# B&R Automation Studio project TD52 (part 16)

```c
/* Source: dspcon.f */
#define dspcon FORTRAN_WRAPPER(dspcon)
extern void dspcon(
    char   *uplo,
    ptrdiff_t *n,
    double *ap,
    ptrdiff_t *ipiv,
    double *anorm,
    double *rcond,
    double *work,
    ptrdiff_t *iwork,
    ptrdiff_t *info
);

/* Source: dspev.f */
#define dspev FORTRAN_WRAPPER(dspev)
extern void dspev(
    char   *jobz,
    char   *uplo,
    ptrdiff_t *n,
    double *ap,
    double *w,
    double *z,
    ptrdiff_t *ldz,
    double *work,
    ptrdiff_t *info
);

/* Source: dspevd.f */
#define dspevd FORTRAN_WRAPPER(dspevd)
extern void dspevd(
    char   *jobz,
    char   *uplo,
    ptrdiff_t *n,
    double *ap,
    double *w,
    double *z,
    ptrdiff_t *ldz,
    double *work,
    ptrdiff_t *lwork,
    ptrdiff_t *iwork,
    ptrdiff_t *liwork,
    ptrdiff_t *info
);

/* Source: dspevx.f */
#define dspevx FORTRAN_WRAPPER(dspevx)
extern void dspevx(
    char   *jobz,
    char   *range,
    char   *uplo,
    ptrdiff_t *n,
    double *ap,
    double *vl,
    double *vu,
    ptrdiff_t *il,
    ptrdiff_t *iu,
    double *abstol,
    ptrdiff_t *m,
    double *w,
    double *z,
    ptrdiff_t *ldz,
    double *work,
    ptrdiff_t *iwork,
    ptrdiff_t *ifail,
    ptrdiff_t *info
);

/* Source: dspgst.f */
#define dspgst FORTRAN_WRAPPER(dspgst)
extern void dspgst(
    ptrdiff_t *itype,
    char   *uplo,
    ptrdiff_t *n,
    double *ap,
    double *bp,
    ptrdiff_t *info
);

/* Source: dspgv.f */
#define dspgv FORTRAN_WRAPPER(dspgv)
extern void dspgv(
    ptrdiff_t *itype,
    char   *jobz,
    char   *uplo,
    ptrdiff_t *n,
    double *ap,
    double *bp,
    double *w,
    double *z,
    ptrdiff_t *ldz,
    double *work,
    ptrdiff_t *info
);

/* Source: dspgvd.f */
#define dspgvd FORTRAN_WRAPPER(dspgvd)
extern void dspgvd(
    ptrdiff_t *itype,
    char   *jobz,
    char   *uplo,
    ptrdiff_t *n,
    double *ap,
    double *bp,
    double *w,
    double *z,
    ptrdiff_t *ldz,
    double *work,
    ptrdiff_t *lwork,
    ptrdiff_t *iwork,
    ptrdiff_t *liwork,
    ptrdiff_t *info
);

/* Source: dspgvx.f */
#define dspgvx FORTRAN_WRAPPER(dspgvx)
extern void dspgvx(
    ptrdiff_t *itype,
    char   *jobz,
    char   *range,
    char   *uplo,
    ptrdiff_t *n,
    double *ap,
    double *bp,
    double *vl,
    double *vu,
    ptrdiff_t *il,
    ptrdiff_t *iu,
    double *abstol,
    ptrdiff_t *m,
    double *w,
    double *z,
    ptrdiff_t *ldz,
    double *work,
    ptrdiff_t *iwork,
    ptrdiff_t *ifail,
    ptrdiff_t *info
);

/* Source: dsposv.f */
#define dsposv FORTRAN_WRAPPER(dsposv)
extern void dsposv(
    char   *uplo,
    ptrdiff_t *n,
    ptrdiff_t *nrhs,
    double *a,
    ptrdiff_t *lda,
    double *b,
    ptrdiff_t *ldb,
    double *x,
    ptrdiff_t *ldx,
    double *work,
    float  *swork,
    ptrdiff_t *iter,
    ptrdiff_t *info
);

/* Source: dsprfs.f */
#define dsprfs FORTRAN_WRAPPER(dsprfs)
extern void dsprfs(
    char   *uplo,
    ptrdiff_t *n,
    ptrdiff_t *nrhs,
    double *ap,
    double *afp,
    ptrdiff_t *ipiv,
    double *b,
    ptrdiff_t *ldb,
    double *x,
    ptrdiff_t *ldx,
    double *ferr,
    double *berr,
    double *work,
    ptrdiff_t *iwork,
    ptrdiff_t *info
);

/* Source: dspsv.f */
#define dspsv FORTRAN_WRAPPER(dspsv)
extern void dspsv(
    char   *uplo,
    ptrdiff_t *n,
    ptrdiff_t *nrhs,
    double *ap,
    ptrdiff_t *ipiv,
    double *b,
    ptrdiff_t *ldb,
    ptrdiff_t *info
);

/* Source: dspsvx.f */
#define dspsvx FORTRAN_WRAPPER(dspsvx)
extern void dspsvx(
    char   *fact,
    char   *uplo,
    ptrdiff_t *n,
    ptrdiff_t *nrhs,
    double *ap,
    double *afp,
    ptrdiff_t *ipiv,
    double *b,
    ptrdiff_t *ldb,
    double *x,
    ptrdiff_t *ldx,
    double *rcond,
    double *ferr,
    double *berr,
    double *work,
    ptrdiff_t *iwork,
    ptrdiff_t *info
);

/* Source: dsptrd.f */
#define dsptrd FORTRAN_WRAPPER(dsptrd)
extern void dsptrd(
    char   *uplo,
    ptrdiff_t *n,
    double *ap,
    double *d,
    double *e,
    double *tau,
    ptrdiff_t *info
);

/* Source: dsptrf.f */
#define dsptrf FORTRAN_WRAPPER(dsptrf)
extern void dsptrf(
    char   *uplo,
    ptrdiff_t *n,
    double *ap,
    ptrdiff_t *ipiv,
    ptrdiff_t *info
);

/* Source: dsptri.f */
#define dsptri FORTRAN_WRAPPER(dsptri)
extern void dsptri(
    char   *uplo,
    ptrdiff_t *n,
    double *ap,
    ptrdiff_t *ipiv,
    double *work,
    ptrdiff_t *info
);

/* Source: dsptrs.f */
#define dsptrs FORTRAN_WRAPPER(dsptrs)
extern void dsptrs(
    char   *uplo,
    ptrdiff_t *n,
    ptrdiff_t *nrhs,
    double *ap,
    ptrdiff_t *ipiv,
    double *b,
    ptrdiff_t *ldb,
    ptrdiff_t *info
);

/* Source: dstebz.f */
#define dstebz FORTRAN_WRAPPER(dstebz)
extern void dstebz(
    char   *range,
    char   *order,
    ptrdiff_t *n,
    double *vl,
    double *vu,
    ptrdiff_t *il,
    ptrdiff_t *iu,
    double *abstol,
    double *d,
    double *e,
    ptrdiff_t *m,
    ptrdiff_t *nsplit,
    double *w,
    ptrdiff_t *iblock,
    ptrdiff_t *isplit,
    double *work,
    ptrdiff_t *iwork,
    ptrdiff_t *info
);

/* Source: dstedc.f */
#define dstedc FORTRAN_WRAPPER(dstedc)
extern void dstedc(
    char   *compz,
    ptrdiff_t *n,
    double *d,
    double *e,
    double *z,
    ptrdiff_t *ldz,
    double *work,
    ptrdiff_t *lwork,
    ptrdiff_t *iwork,
    ptrdiff_t *liwork,
    ptrdiff_t *info
);

/* Source: dstegr.f */
#define dstegr FORTRAN_WRAPPER(dstegr)
extern void dstegr(
    char   *jobz,
    char   *range,
    ptrdiff_t *n,
    double *d,
    double *e,
    double *vl,
    double *vu,
    ptrdiff_t *il,
    ptrdiff_t *iu,
    double *abstol,
    ptrdiff_t *m,
    double *w,
    double *z,
    ptrdiff_t *ldz,
    ptrdiff_t *isuppz,
    double *work,
    ptrdiff_t *lwork,
    ptrdiff_t *iwork,
    ptrdiff_t *liwork,
    ptrdiff_t *info
);

/* Source: dstein.f */
#define dstein FORTRAN_WRAPPER(dstein)
extern void dstein(
    ptrdiff_t *n,
    double *d,
    double *e,
    ptrdiff_t *m,
    double *w,
    ptrdiff_t *iblock,
    ptrdiff_t *isplit,
    double *z,
    ptrdiff_t *ldz,
    double *work,
    ptrdiff_t *iwork,
    ptrdiff_t *ifail,
    ptrdiff_t *info
);

/* Source: dstemr.f */
#define dstemr FORTRAN_WRAPPER(dstemr)
extern void dstemr(
    char   *jobz,
    char   *range,
    ptrdiff_t *n,
    double *d,
    double *e,
    double *vl,
    double *vu,
    ptrdiff_t *il,
    ptrdiff_t *iu,
    ptrdiff_t *m,
    double *w,
    double *z,
    ptrdiff_t *ldz,
    ptrdiff_t *nzc,
    ptrdiff_t *isuppz,
    ptrdiff_t *tryrac,
    double *work,
    ptrdiff_t *lwork,
    ptrdiff_t *iwork,
    ptrdiff_t *liwork,
    ptrdiff_t *info
);

/* Source: dsteqr.f */
#define dsteqr FORTRAN_WRAPPER(dsteqr)
extern void dsteqr(
    char   *compz,
    ptrdiff_t *n,
    double *d,
    double *e,
    double *z,
    ptrdiff_t *ldz,
    double *work,
    ptrdiff_t *info
);

/* Source: dsterf.f */
#define dsterf FORTRAN_WRAPPER(dsterf)
extern void dsterf(
    ptrdiff_t *n,
    double *d,
    double *e,
    ptrdiff_t *info
);

/* Source: dstev.f */
#define dstev FORTRAN_WRAPPER(dstev)
extern void dstev(
    char   *jobz,
    ptrdiff_t *n,
    double *d,
    double *e,
    double *z,
    ptrdiff_t *ldz,
    double *work,
    ptrdiff_t *info
);

/* Source: dstevd.f */
#define dstevd FORTRAN_WRAPPER(dstevd)
extern void dstevd(
    char   *jobz,
    ptrdiff_t *n,
    double *d,
    double *e,
    double *z,
    ptrdiff_t *ldz,
    double *work,
    ptrdiff_t *lwork,
    ptrdiff_t *iwork,
    ptrdiff_t *liwork,
    ptrdiff_t *info
);

/* Source: dstevr.f */
#define dstevr FORTRAN_WRAPPER(dstevr)
extern void dstevr(
    char   *jobz,
    char   *range,
    ptrdiff_t *n,
    double *d,
    double *e,
    double *vl,
    double *vu,
    ptrdiff_t *il,
    ptrdiff_t *iu,
    double *abstol,
    ptrdiff_t *m,
    double *w,
    double *z,
    ptrdiff_t *ldz,
    ptrdiff_t *isuppz,
    double *work,
    ptrdiff_t *lwork,
    ptrdiff_t *iwork,
    ptrdiff_t *liwork,
    ptrdiff_t *info
);

/* Source: dstevx.f */
#define dstevx FORTRAN_WRAPPER(dstevx)
extern void dstevx(
    char   *jobz,
    char   *range,
    ptrdiff_t *n,
    double *d,
    double *e,
    double *vl,
    double *vu,
    ptrdiff_t *il,
    ptrdiff_t *iu,
    double *abstol,
    ptrdiff_t *m,
    double *w,
    double *z,
    ptrdiff_t *ldz,
    double *work,
    ptrdiff_t *iwork,
    ptrdiff_t *ifail,
    ptrdiff_t *info
);

/* Source: dsycon.f */
#define dsycon FORTRAN_WRAPPER(dsycon)
extern void dsycon(
    char   *uplo,
    ptrdiff_t *n,
    double *a,
    ptrdiff_t *lda,
    ptrdiff_t *ipiv,
    double *anorm,
    double *rcond,
    double *work,
    ptrdiff_t *iwork,
    ptrdiff_t *info
);

/* Source: dsyequb.f */
#define dsyequb FORTRAN_WRAPPER(dsyequb)
extern void dsyequb(
    char   *uplo,
    ptrdiff_t *n,
    double *a,
    ptrdiff_t *lda,
    double *s,
    double *scond,
    double *amax,
    double *work,
    ptrdiff_t *info
);

/* Source: dsyev.f */
#define dsyev FORTRAN_WRAPPER(dsyev)
extern void dsyev(
    char   *jobz,
    char   *uplo,
    ptrdiff_t *n,
    double *a,
    ptrdiff_t *lda,
    double *w,
    double *work,
    ptrdiff_t *lwork,
    ptrdiff_t *info
);

/* Source: dsyevd.f */
#define dsyevd FORTRAN_WRAPPER(dsyevd)
extern void dsyevd(
    char   *jobz,
    char   *uplo,
    ptrdiff_t *n,
    double *a,
    ptrdiff_t *lda,
    double *w,
    double *work,
    ptrdiff_t *lwork,
    ptrdiff_t *iwork,
    ptrdiff_t *liwork,
    ptrdiff_t *info
);

/* Source: dsyevr.f */
#define dsyevr FORTRAN_WRAPPER(dsyevr)
extern void dsyevr(
    char   *jobz,
    char   *range,
    char   *uplo,
    ptrdiff_t *n,
    double *a,
    ptrdiff_t *lda,
    double *vl,
    double *vu,
    ptrdiff_t *il,
    ptrdiff_t *iu,
    double *abstol,
    ptrdiff_t *m,
    double *w,
    double *z,
    ptrdiff_t *ldz,
    ptrdiff_t *isuppz,
    double *work,
    ptrdiff_t *lwork,
    ptrdiff_t *iwork,
    ptrdiff_t *liwork,
    ptrdiff_t *info
);

/* Source: dsyevx.f */
#define dsyevx FORTRAN_WRAPPER(dsyevx)
extern void dsyevx(
    char   *jobz,
    char   *range,
    char   *uplo,
    ptrdiff_t *n,
    double *a,
    ptrdiff_t *lda,
    double *vl,
    double *vu,
    ptrdiff_t *il,
    ptrdiff_t *iu,
    double *abstol,
    ptrdiff_t *m,
    double *w,
    double *z,
    ptrdiff_t *ldz,
    double *work,
    ptrdiff_t *lwork,
    ptrdiff_t *iwork,
    ptrdiff_t *ifail,
    ptrdiff_t *info
);

/* Source: dsygs2.f */
#define dsygs2 FORTRAN_WRAPPER(dsygs2)
extern void dsygs2(
    ptrdiff_t *itype,
    char   *uplo,
    ptrdiff_t *n,
    double *a,
    ptrdiff_t *lda,
    double *b,
    ptrdiff_t *ldb,
    ptrdiff_t *info
);

/* Source: dsygst.f */
#define dsygst FORTRAN_WRAPPER(dsygst)
extern void dsygst(
    ptrdiff_t *itype,
    char   *uplo,
    ptrdiff_t *n,
    double *a,
    ptrdiff_t *lda,
    double *b,
    ptrdiff_t *ldb,
    ptrdiff_t *info
);

/* Source: dsygv.f */
#define dsygv FORTRAN_WRAPPER(dsygv)
extern void dsygv(
    ptrdiff_t *itype,
    char   *jobz,
    char   *uplo,
    ptrdiff_t *n,
    double *a,
    ptrdiff_t *lda,
    double *b,
    ptrdiff_t *ldb,
    double *w,
    double *work,
    ptrdiff_t *lwork,
    ptrdiff_t *info
);

/* Source: dsygvd.f */
#define dsygvd FORTRAN_WRAPPER(dsygvd)
extern void dsygvd(
    ptrdiff_t *itype,
    char   *jobz,
    char   *uplo,
    ptrdiff_t *n,
    double *a,
    ptrdiff_t *lda,
    double *b,
    ptrdiff_t *ldb,
    double *w,
    double *work,
    ptrdiff_t *lwork,
    ptrdiff_t *iwork,
    ptrdiff_t *liwork,
    ptrdiff_t *info
);

/* Source: dsygvx.f */
#define dsygvx FORTRAN_WRAPPER(dsygvx)
extern void dsygvx(
    ptrdiff_t *itype,
    char   *jobz,
    char   *range,
    char   *uplo,
    ptrdiff_t *n,
    double *a,
    ptrdiff_t *lda,
    double *b,
    ptrdiff_t *ldb,
    double *vl,
    double *vu,
    ptrdiff_t *il,
    ptrdiff_t *iu,
    double *abstol,
    ptrdiff_t *m,
    double *w,
    double *z,
    ptrdiff_t *ldz,
    double *work,
    ptrdiff_t *lwork,
    ptrdiff_t *iwork,
    ptrdiff_t *ifail,
    ptrdiff_t *info
);

/* Source: dsyrfs.f */
#define dsyrfs FORTRAN_WRAPPER(dsyrfs)
extern void dsyrfs(
    char   *uplo,
    ptrdiff_t *n,
    ptrdiff_t *nrhs,
    double *a,
    ptrdiff_t *lda,
    double *af,
    ptrdiff_t *ldaf,
    ptrdiff_t *ipiv,
    double *b,
    ptrdiff_t *ldb,
    double *x,
    ptrdiff_t *ldx,
    double *ferr,
    double *berr,
    double *work,
    ptrdiff_t *iwork,
    ptrdiff_t *info
);

/* Source: dsysv.f */
#define dsysv FORTRAN_WRAPPER(dsysv)
extern void dsysv(
    char   *uplo,
    ptrdiff_t *n,
    ptrdiff_t *nrhs,
    double *a,
    ptrdiff_t *lda,
    ptrdiff_t *ipiv,
    double *b,
    ptrdiff_t *ldb,
    double *work,
    ptrdiff_t *lwork,
    ptrdiff_t *info
);

/* Source: dsysvx.f */
#define dsysvx FORTRAN_WRAPPER(dsysvx)
extern void dsysvx(
    char   *fact,
    char   *uplo,
    ptrdiff_t *n,
    ptrdiff_t *nrhs,
    double *a,
    ptrdiff_t *lda,
    double *af,
    ptrdiff_t *ldaf,
    ptrdiff_t *ipiv,
    double *b,
    ptrdiff_t *ldb,
    double *x,
    ptrdiff_t *ldx,
    double *rcond,
    double *ferr,
    double *berr,
    double *work,
    ptrdiff_t *lwork,
    ptrdiff_t *iwork,
    ptrdiff_t *info
);

/* Source: dsytd2.f */
#define dsytd2 FORTRAN_WRAPPER(dsytd2)
extern void dsytd2(
    char   *uplo,
    ptrdiff_t *n,
    double *a,
    ptrdiff_t *lda,
    double *d,
    double *e,
    double *tau,
    ptrdiff_t *info
);

/* Source: dsytf2.f */
#define dsytf2 FORTRAN_WRAPPER(dsytf2)
extern void dsytf2(
    char   *uplo,
    ptrdiff_t *n,
    double *a,
    ptrdiff_t *lda,
    ptrdiff_t *ipiv,
    ptrdiff_t *info
);

/* Source: dsytrd.f */
#define dsytrd FORTRAN_WRAPPER(dsytrd)
extern void dsytrd(
    char   *uplo,
    ptrdiff_t *n,
    double *a,
    ptrdiff_t *lda,
    double *d,
    double *e,
    double *tau,
    double *work,
    ptrdiff_t *lwork,
    ptrdiff_t *info
);

/* Source: dsytrf.f */
#define dsytrf FORTRAN_WRAPPER(dsytrf)
extern void dsytrf(
    char   *uplo,
    ptrdiff_t *n,
    double *a,
    ptrdiff_t *lda,
    ptrdiff_t *ipiv,
    double *work,
    ptrdiff_t *lwork,
    ptrdiff_t *info
);

/* Source: dsytri.f */
#define dsytri FORTRAN_WRAPPER(dsytri)
extern void dsytri(
    char   *uplo,
    ptrdiff_t *n,
    double *a,
    ptrdiff_t *lda,
    ptrdiff_t *ipiv,
    double *work,
    ptrdiff_t *info
);

/* Source: dsytrs.f */
#define dsytrs FORTRAN_WRAPPER(dsytrs)
extern void dsytrs(
    char   *uplo,
    ptrdiff_t *n,
    ptrdiff_t *nrhs,
    double *a,
    ptrdiff_t *lda,
    ptrdiff_t *ipiv,
    double *b,
    ptrdiff_t *ldb,
    ptrdiff_t *info
);

/* Source: dtbcon.f */
#define dtbcon FORTRAN_WRAPPER(dtbcon)
extern void dtbcon(
    char   *norm,
    char   *uplo,
    char   *diag,
    ptrdiff_t *n,
    ptrdiff_t *kd,
    double *ab,
    ptrdiff_t *ldab,
    double *rcond,
    double *work,
    ptrdiff_t *iwork,
    ptrdiff_t *info
);

/* Source: dtbrfs.f */
#define dtbrfs FORTRAN_WRAPPER(dtbrfs)
extern void dtbrfs(
    char   *uplo,
    char   *trans,
    char   *diag,
    ptrdiff_t *n,
    ptrdiff_t *kd,
    ptrdiff_t *nrhs,
    double *ab,
    ptrdiff_t *ldab,
    double *b,
    ptrdiff_t *ldb,
    double *x,
    ptrdiff_t *ldx,
    double *ferr,
    double *berr,
    double *work,
    ptrdiff_t *iwork,
    ptrdiff_t *info
);

/* Source: dtbtrs.f */
#define dtbtrs FORTRAN_WRAPPER(dtbtrs)
extern void dtbtrs(
    char   *uplo,
    char   *trans,
    char   *diag,
    ptrdiff_t *n,
    ptrdiff_t *kd,
    ptrdiff_t *nrhs,
    double *ab,
    ptrdiff_t *ldab,
    double *b,
    ptrdiff_t *ldb,
    ptrdiff_t *info
);

/* Source: dtfsm.f */
#define dtfsm FORTRAN_WRAPPER(dtfsm)
extern void dtfsm(
    char   *transr,
    char   *side,
    char   *uplo,
    char   *trans,
    char   *diag,
    ptrdiff_t *m,
    ptrdiff_t *n,
    double *alpha,
    double *a,
    double *b,
    ptrdiff_t *ldb
);

/* Source: dtftri.f */
#define dtftri FORTRAN_WRAPPER(dtftri)
extern void dtftri(
    char   *transr,
    char   *uplo,
    char   *diag,
    ptrdiff_t *n,
    double *a,
    ptrdiff_t *info
);

/* Source: dtfttp.f */
#define dtfttp FORTRAN_WRAPPER(dtfttp)
extern void dtfttp(
    char   *transr,
    char   *uplo,
    ptrdiff_t *n,
    double *arf,
    double *ap,
    ptrdiff_t *info
);

/* Source: dtfttr.f */
#define dtfttr FORTRAN_WRAPPER(dtfttr)
extern void dtfttr(
    char   *transr,
    char   *uplo,
    ptrdiff_t *n,
    double *arf,
    double *a,
    ptrdiff_t *lda,
    ptrdiff_t *info
);

/* Source: dtgevc.f */
#define dtgevc FORTRAN_WRAPPER(dtgevc)
extern void dtgevc(
    char   *side,
    char   *howmny,
    ptrdiff_t *select,
    ptrdiff_t *n,
    double *s,
    ptrdiff_t *lds,
    double *p,
    ptrdiff_t *ldp,
    double *vl,
    ptrdiff_t *ldvl,
    double *vr,
    ptrdiff_t *ldvr,
    ptrdiff_t *mm,
    ptrdiff_t *m,
    double *work,
    ptrdiff_t *info
);

/* Source: dtgex2.f */
#define dtgex2 FORTRAN_WRAPPER(dtgex2)
extern void dtgex2(
    ptrdiff_t *wantq,
    ptrdiff_t *wantz,
    ptrdiff_t *n,
    double *a,
    ptrdiff_t *lda,
    double *b,
    ptrdiff_t *ldb,
    double *q,
    ptrdiff_t *ldq,
    double *z,
    ptrdiff_t *ldz,
    ptrdiff_t *j1_,
    ptrdiff_t *n1,
    ptrdiff_t *n2,
    double *work,
    ptrdiff_t *lwork,
    ptrdiff_t *info
);

/* Source: dtgexc.f */
#define dtgexc FORTRAN_WRAPPER(dtgexc)
extern void dtgexc(
    ptrdiff_t *wantq,
    ptrdiff_t *wantz,
    ptrdiff_t *n,
    double *a,
    ptrdiff_t *lda,
    double *b,
    ptrdiff_t *ldb,
    double *q,
    ptrdiff_t *ldq,
    double *z,
    ptrdiff_t *ldz,
    ptrdiff_t *ifst,
    ptrdiff_t *ilst,
    double *work,
    ptrdiff_t *lwork,
    ptrdiff_t *info
);

/* Source: dtgsen.f */
#define dtgsen FORTRAN_WRAPPER(dtgsen)
extern void dtgsen(
    ptrdiff_t *ijob,
    ptrdiff_t *wantq,
    ptrdiff_t *wantz,
    ptrdiff_t *select,
    ptrdiff_t *n,
    double *a,
    ptrdiff_t *lda,
    double *b,
    ptrdiff_t *ldb,
    double *alphar,
    double *alphai,
    double *beta,
    double *q,
    ptrdiff_t *ldq,
    double *z,
    ptrdiff_t *ldz,
    ptrdiff_t *m,
    double *pl,
    double *pr,
    double *dif,
    double *work,
    ptrdiff_t *lwork,
    ptrdiff_t *iwork,
    ptrdiff_t *liwork,
    ptrdiff_t *info
);

/* Source: dtgsja.f */
#define dtgsja FORTRAN_WRAPPER(dtgsja)
extern void dtgsja(
    char   *jobu,
    char   *jobv,
    char   *jobq,
    ptrdiff_t *m,
    ptrdiff_t *p,
    ptrdiff_t *n,
    ptrdiff_t *k,
    ptrdiff_t *l,
    double *a,
    ptrdiff_t *lda,
    double *b,
    ptrdiff_t *ldb,
    double *tola,
    double *tolb,
    double *alpha,
    double *beta,
    double *u,
    ptrdiff_t *ldu,
    double *v,
    ptrdiff_t *ldv,
    double *q,
    ptrdiff_t *ldq,
    double *work,
    ptrdiff_t *ncycle,
    ptrdiff_t *info
);

/* Source: dtgsna.f */
#define dtgsna FORTRAN_WRAPPER(dtgsna)
extern void dtgsna(
    char   *job,
    char   *howmny,
    ptrdiff_t *select,
    ptrdiff_t *n,
    double *a,
    ptrdiff_t *lda,
    double *b,
    ptrdiff_t *ldb,
    double *vl,
    ptrdiff_t *ldvl,
    double *vr,
    ptrdiff_t *ldvr,
    double *s,
    double *dif,
    ptrdiff_t *mm,
    ptrdiff_t *m,
    double *work,
    ptrdiff_t *lwork,
    ptrdiff_t *iwork,
    ptrdiff_t *info
);

/* Source: dtgsy2.f */
#define dtgsy2 FORTRAN_WRAPPER(dtgsy2)
extern void dtgsy2(
    char   *trans,
    ptrdiff_t *ijob,
    ptrdiff_t *m,
    ptrdiff_t *n,
    double *a,
    ptrdiff_t *lda,
    double *b,
    ptrdiff_t *ldb,
    double *c,
    ptrdiff_t *ldc,
    double *d,
    ptrdiff_t *ldd,
    double *e,
    ptrdiff_t *lde,
    double *f,
    ptrdiff_t *ldf,
    double *scale,
    double *rdsum,
    double *rdscal,
    ptrdiff_t *iwork,
    ptrdiff_t *pq,
    ptrdiff_t *info
);

/* Source: dtgsyl.f */
#define dtgsyl FORTRAN_WRAPPER(dtgsyl)
extern void dtgsyl(
    char   *trans,
    ptrdiff_t *ijob,
    ptrdiff_t *m,
    ptrdiff_t *n,
    double *a,
    ptrdiff_t *lda,
    double *b,
    ptrdiff_t *ldb,
    double *c,
    ptrdiff_t *ldc,
    double *d,
    ptrdiff_t *ldd,
    double *e,
    ptrdiff_t *lde,
    double *f,
    ptrdiff_t *ldf,
    double *scale,
    double *dif,
    double *work,
    ptrdiff_t *lwork,
    ptrdiff_t *iwork,
    ptrdiff_t *info
);

/* Source: dtpcon.f */
#define dtpcon FORTRAN_WRAPPER(dtpcon)
extern void dtpcon(
    char   *norm,
    char   *uplo,
    char   *diag,
    ptrdiff_t *n,
    double *ap,
    double *rcond,
    double *work,
    ptrdiff_t *iwork,
    ptrdiff_t *info
);

/* Source: dtprfs.f */
#define dtprfs FORTRAN_WRAPPER(dtprfs)
extern void dtprfs(
    char   *uplo,
    char   *trans,
    char   *diag,
    ptrdiff_t *n,
    ptrdiff_t *nrhs,
    double *ap,
    double *b,
    ptrdiff_t *ldb,
    double *x,
    ptrdiff_t *ldx,
    double *ferr,
    double *berr,
    double *work,
    ptrdiff_t *iwork,
    ptrdiff_t *info
);

/* Source: dtptri.f */
#define dtptri FORTRAN_WRAPPER(dtptri)
extern void dtptri(
    char   *uplo,
    char   *diag,
    ptrdiff_t *n,
    double *ap,
    ptrdiff_t *info
);

/* Source: dtptrs.f */
#define dtptrs FORTRAN_WRAPPER(dtptrs)
extern void dtptrs(
    char   *uplo,
    char   *trans,
    char   *diag,
    ptrdiff_t *n,
    ptrdiff_t *nrhs,
    double *ap,
    double *b,
    ptrdiff_t *ldb,
    ptrdiff_t *info
);

/* Source: dtpttf.f */
#define dtpttf FORTRAN_WRAPPER(dtpttf)
extern void dtpttf(
    char   *transr,
    char   *uplo,
    ptrdiff_t *n,
    double *ap,
    double *arf,
    ptrdiff_t *info
);

/* Source: dtpttr.f */
#define dtpttr FORTRAN_WRAPPER(dtpttr)
extern void dtpttr(
    char   *uplo,
    ptrdiff_t *n,
    double *ap,
    double *a,
    ptrdiff_t *lda,
    ptrdiff_t *info
);

/* Source: dtrcon.f */
#define dtrcon FORTRAN_WRAPPER(dtrcon)
extern void dtrcon(
    char   *norm,
    char   *uplo,
    char   *diag,
    ptrdiff_t *n,
    double *a,
    ptrdiff_t *lda,
    double *rcond,
    double *work,
    ptrdiff_t *iwork,
    ptrdiff_t *info
);

/* Source: dtrevc.f */
#define dtrevc FORTRAN_WRAPPER(dtrevc)
extern void dtrevc(
    char   *side,
    char   *howmny,
    ptrdiff_t *select,
    ptrdiff_t *n,
    double *t,
    ptrdiff_t *ldt,
    double *vl,
    ptrdiff_t *ldvl,
    double *vr,
    ptrdiff_t *ldvr,
    ptrdiff_t *mm,
    ptrdiff_t *m,
    double *work,
    ptrdiff_t *info
);

/* Source: dtrexc.f */
#define dtrexc FORTRAN_WRAPPER(dtrexc)
extern void dtrexc(
    char   *compq,
    ptrdiff_t *n,
    double *t,
    ptrdiff_t *ldt,
    double *q,
    ptrdiff_t *ldq,
    ptrdiff_t *ifst,
    ptrdiff_t *ilst,
    double *work,
    ptrdiff_t *info
);

/* Source: dtrrfs.f */
#define dtrrfs FORTRAN_WRAPPER(dtrrfs)
extern void dtrrfs(
    char   *uplo,
    char   *trans,
    char   *diag,
    ptrdiff_t *n,
    ptrdiff_t *nrhs,
    double *a,
    ptrdiff_t *lda,
    double *b,
    ptrdiff_t *ldb,
    double *x,
    ptrdiff_t *ldx,
    double *ferr,
    double *berr,
    double *work,
    ptrdiff_t *iwork,
    ptrdiff_t *info
);

/* Source: dtrsen.f */
#define dtrsen FORTRAN_WRAPPER(dtrsen)
extern void dtrsen(
    char   *job,
    char   *compq,
    ptrdiff_t *select,
    ptrdiff_t *n,
    double *t,
    ptrdiff_t *ldt,
    double *q,
    ptrdiff_t *ldq,
    double *wr,
    double *wi,
    ptrdiff_t *m,
    double *s,
    double *sep,
    double *work,
    ptrdiff_t *lwork,
    ptrdiff_t *iwork,
    ptrdiff_t *liwork,
    ptrdiff_t *info
);

/* Source: dtrsna.f */
#define dtrsna FORTRAN_WRAPPER(dtrsna)
extern void dtrsna(
    char   *job,
    char   *howmny,
    ptrdiff_t *select,
    ptrdiff_t *n,
    double *t,
    ptrdiff_t *ldt,
    double *vl,
    ptrdiff_t *ldvl,
    double *vr,
    ptrdiff_t *ldvr,
    double *s,
    double *sep,
    ptrdiff_t *mm,
    ptrdiff_t *m,
    double *work,
    ptrdiff_t *ldwork,
    ptrdiff_t *iwork,
    ptrdiff_t *info
);

/* Source: dtrsyl.f */
#define dtrsyl FORTRAN_WRAPPER(dtrsyl)
extern void dtrsyl(
    char   *trana,
    char   *tranb,
    ptrdiff_t *isgn,
    ptrdiff_t *m,
    ptrdiff_t *n,
    double *a,
    ptrdiff_t *lda,
    double *b,
    ptrdiff_t *ldb,
    double *c,
    ptrdiff_t *ldc,
    double *scale,
    ptrdiff_t *info
);

/* Source: dtrti2.f */
#define dtrti2 FORTRAN_WRAPPER(dtrti2)
extern void dtrti2(
    char   *uplo,
    char   *diag,
    ptrdiff_t *n,
    double *a,
    ptrdiff_t *lda,
    ptrdiff_t *info
);

/* Source: dtrtri.f */
#define dtrtri FORTRAN_WRAPPER(dtrtri)
extern void dtrtri(
    char   *uplo,
    char   *diag,
    ptrdiff_t *n,
    double *a,
    ptrdiff_t *lda,
    ptrdiff_t *info
);

/* Source: dtrtrs.f */
#define dtrtrs FORTRAN_WRAPPER(dtrtrs)
extern void dtrtrs(
    char   *uplo,
    char   *trans,
    char   *diag,
    ptrdiff_t *n,
    ptrdiff_t *nrhs,
    double *a,
    ptrdiff_t *lda,
    double *b,
    ptrdiff_t *ldb,
    ptrdiff_t *info
);

/* Source: dtrttf.f */
#define dtrttf FORTRAN_WRAPPER(dtrttf)
extern void dtrttf(
    char   *transr,
    char   *uplo,
    ptrdiff_t *n,
    double *a,
    ptrdiff_t *lda,
    double *arf,
    ptrdiff_t *info
);

/* Source: dtrttp.f */
#define dtrttp FORTRAN_WRAPPER(dtrttp)
extern void dtrttp(
    char   *uplo,
    ptrdiff_t *n,
    double *a,
    ptrdiff_t *lda,
    double *ap,
    ptrdiff_t *info
);

/* Source: dtzrqf.f */
#define dtzrqf FORTRAN_WRAPPER(dtzrqf)
extern void dtzrqf(
    ptrdiff_t *m,
    ptrdiff_t *n,
    double *a,
    ptrdiff_t *lda,
    double *tau,
    ptrdiff_t *info
);

/* Source: dtzrzf.f */
#define dtzrzf FORTRAN_WRAPPER(dtzrzf)
extern void dtzrzf(
    ptrdiff_t *m,
    ptrdiff_t *n,
    double *a,
    ptrdiff_t *lda,
    double *tau,
    double *work,
    ptrdiff_t *lwork,
    ptrdiff_t *info
);

/* Source: dzsum1.f */
#define dzsum1 FORTRAN_WRAPPER(dzsum1)
extern double dzsum1(
    ptrdiff_t *n,
    double *cx,
    ptrdiff_t *incx
);

/* Source: icmax1.f */
#define icmax1 FORTRAN_WRAPPER(icmax1)
extern ptrdiff_t icmax1(
    ptrdiff_t *n,
    float  *cx,
    ptrdiff_t *incx
);

/* Source: ieeeck.f */
#define ieeeck FORTRAN_WRAPPER(ieeeck)
extern ptrdiff_t ieeeck(
    ptrdiff_t *ispec,
    float  *zero,
    float  *one
);

/* Source: ilaclc.f */
#define ilaclc FORTRAN_WRAPPER(ilaclc)
extern ptrdiff_t ilaclc(
    ptrdiff_t *m,
    ptrdiff_t *n,
    float  *a,
    ptrdiff_t *lda
);

/* Source: ilaclr.f */
#define ilaclr FORTRAN_WRAPPER(ilaclr)
extern ptrdiff_t ilaclr(
    ptrdiff_t *m,
    ptrdiff_t *n,
    float  *a,
    ptrdiff_t *lda
);

/* Source: iladiag.f */
#define iladiag FORTRAN_WRAPPER(iladiag)
extern ptrdiff_t iladiag(
    char   *diag
);

/* Source: iladlc.f */
#define iladlc FORTRAN_WRAPPER(iladlc)
extern ptrdiff_t iladlc(
    ptrdiff_t *m,
    ptrdiff_t *n,
    double *a,
    ptrdiff_t *lda
);

/* Source: iladlr.f */
#define iladlr FORTRAN_WRAPPER(iladlr)
extern ptrdiff_t iladlr(
    ptrdiff_t *m,
    ptrdiff_t *n,
    double *a,
    ptrdiff_t *lda
);

/* Source: ilaenv.f */
#define ilaenv FORTRAN_WRAPPER(ilaenv)
extern ptrdiff_t ilaenv(
    ptrdiff_t *ispec,
    char   *name,
    char   *opts,
    ptrdiff_t *n1,
    ptrdiff_t *n2,
    ptrdiff_t *n3,
    ptrdiff_t *n4,
    ptrdiff_t name_len,
    ptrdiff_t opts_len
);

/* Source: ilaprec.f */
#define ilaprec FORTRAN_WRAPPER(ilaprec)
extern ptrdiff_t ilaprec(
    char   *prec
);

/* Source: ilaslc.f */
#define ilaslc FORTRAN_WRAPPER(ilaslc)
extern ptrdiff_t ilaslc(
    ptrdiff_t *m,
    ptrdiff_t *n,
    float  *a,
    ptrdiff_t *lda
);

/* Source: ilaslr.f */
#define ilaslr FORTRAN_WRAPPER(ilaslr)
extern ptrdiff_t ilaslr(
    ptrdiff_t *m,
    ptrdiff_t *n,
    float  *a,
    ptrdiff_t *lda
);

/* Source: ilatrans.f */
#define ilatrans FORTRAN_WRAPPER(ilatrans)
extern ptrdiff_t ilatrans(
    char   *trans
);

/* Source: ilauplo.f */
#define ilauplo FORTRAN_WRAPPER(ilauplo)
extern ptrdiff_t ilauplo(
    char   *uplo
);

/* Source: ilaver.f */
#define ilaver FORTRAN_WRAPPER(ilaver)
extern void ilaver(
    ptrdiff_t *vers_major,
    ptrdiff_t *vers_minor,
    ptrdiff_t *vers_patch
);

/* Source: ilazlc.f */
#define ilazlc FORTRAN_WRAPPER(ilazlc)
extern ptrdiff_t ilazlc(
    ptrdiff_t *m,
    ptrdiff_t *n,
    double *a,
    ptrdiff_t *lda
);

/* Source: ilazlr.f */
#define ilazlr FORTRAN_WRAPPER(ilazlr)
extern ptrdiff_t ilazlr(
    ptrdiff_t *m,
    ptrdiff_t *n,
    double *a,
    ptrdiff_t *lda
);

/* Source: iparmq.f */
#define iparmq FORTRAN_WRAPPER(iparmq)
extern ptrdiff_t iparmq(
    ptrdiff_t *ispec,
    char   *name,
    char   *opts,
    ptrdiff_t *n,
    ptrdiff_t *ilo,
    ptrdiff_t *ihi,
    ptrdiff_t *lwork
);

/* Source: izmax1.f */
#define izmax1 FORTRAN_WRAPPER(izmax1)
extern ptrdiff_t izmax1(
    ptrdiff_t *n,
    double *cx,
    ptrdiff_t *incx
);

/* Source: lsamen.f */
#define lsamen FORTRAN_WRAPPER(lsamen)
extern ptrdiff_t lsamen(
    ptrdiff_t *n,
    char   *ca,
    char   *cb,
    ptrdiff_t ca_len,
    ptrdiff_t cb_len
);

/* Source: sbdsdc.f */
#define sbdsdc FORTRAN_WRAPPER(sbdsdc)
extern void sbdsdc(
    char   *uplo,
    char   *compq,
    ptrdiff_t *n,
    float  *d,
    float  *e,
    float  *u,
    ptrdiff_t *ldu,
    float  *vt,
    ptrdiff_t *ldvt,
    float  *q,
    ptrdiff_t *iq,
    float  *work,
    ptrdiff_t *iwork,
    ptrdiff_t *info
);

/* Source: sbdsqr.f */
#define sbdsqr FORTRAN_WRAPPER(sbdsqr)
extern void sbdsqr(
    char   *uplo,
    ptrdiff_t *n,
    ptrdiff_t *ncvt,
    ptrdiff_t *nru,
    ptrdiff_t *ncc,
    float  *d,
    float  *e,
    float  *vt,
    ptrdiff_t *ldvt,
    float  *u,
    ptrdiff_t *ldu,
    float  *c,
    ptrdiff_t *ldc,
    float  *work,
    ptrdiff_t *info
);

/* Source: scsum1.f */
#define scsum1 FORTRAN_WRAPPER(scsum1)
#ifdef FORTRAN_FLOAT_FUNCTIONS_RETURN_DOUBLE
extern double scsum1(
#else
extern float scsum1(
#endif
    ptrdiff_t *n,
    float  *cx,
    ptrdiff_t *incx
);

/* Source: sdisna.f */
#define sdisna FORTRAN_WRAPPER(sdisna)
extern void sdisna(
    char   *job,
    ptrdiff_t *m,
    ptrdiff_t *n,
    float  *d,
    float  *sep,
    ptrdiff_t *info
);

/* Source: sgbbrd.f */
#define sgbbrd FORTRAN_WRAPPER(sgbbrd)
extern void sgbbrd(
    char   *vect,
    ptrdiff_t *m,
    ptrdiff_t *n,
    ptrdiff_t *ncc,
    ptrdiff_t *kl,
    ptrdiff_t *ku,
    float  *ab,
    ptrdiff_t *ldab,
    float  *d,
    float  *e,
    float  *q,
    ptrdiff_t *ldq,
    float  *pt,
    ptrdiff_t *ldpt,
    float  *c,
    ptrdiff_t *ldc,
    float  *work,
    ptrdiff_t *info
);

/* Source: sgbcon.f */
#define sgbcon FORTRAN_WRAPPER(sgbcon)
extern void sgbcon(
    char   *norm,
    ptrdiff_t *n,
    ptrdiff_t *kl,
    ptrdiff_t *ku,
    float  *ab,
    ptrdiff_t *ldab,
    ptrdiff_t *ipiv,
    float  *anorm,
    float  *rcond,
    float  *work,
    ptrdiff_t *iwork,
    ptrdiff_t *info
);

/* Source: sgbequ.f */
#define sgbequ FORTRAN_WRAPPER(sgbequ)
extern void sgbequ(
    ptrdiff_t *m,
    ptrdiff_t *n,
    ptrdiff_t *kl,
    ptrdiff_t *ku,
    float  *ab,
    ptrdiff_t *ldab,
    float  *r,
    float  *c,
    float  *rowcnd,
    float  *colcnd,
    float  *amax,
    ptrdiff_t *info
);

/* Source: sgbequb.f */
#define sgbequb FORTRAN_WRAPPER(sgbequb)
extern void sgbequb(
    ptrdiff_t *m,
    ptrdiff_t *n,
    ptrdiff_t *kl,
    ptrdiff_t *ku,
    float  *ab,
    ptrdiff_t *ldab,
    float  *r,
    float  *c,
    float  *rowcnd,
    float  *colcnd,
    float  *amax,
    ptrdiff_t *info
);

/* Source: sgbrfs.f */
#define sgbrfs FORTRAN_WRAPPER(sgbrfs)
extern void sgbrfs(
    char   *trans,
    ptrdiff_t *n,
    ptrdiff_t *kl,
    ptrdiff_t *ku,
    ptrdiff_t *nrhs,
    float  *ab,
    ptrdiff_t *ldab,
    float  *afb,
    ptrdiff_t *ldafb,
    ptrdiff_t *ipiv,
    float  *b,
    ptrdiff_t *ldb,
    float  *x,
    ptrdiff_t *ldx,
    float  *ferr,
    float  *berr,
    float  *work,
    ptrdiff_t *iwork,
    ptrdiff_t *info
);

/* Source: sgbsv.f */
#define sgbsv FORTRAN_WRAPPER(sgbsv)
extern void sgbsv(
    ptrdiff_t *n,
    ptrdiff_t *kl,
    ptrdiff_t *ku,
    ptrdiff_t *nrhs,
    float  *ab,
    ptrdiff_t *ldab,
    ptrdiff_t *ipiv,
    float  *b,
    ptrdiff_t *ldb,
    ptrdiff_t *info
);

/* Source: sgbsvx.f */
#define sgbsvx FORTRAN_WRAPPER(sgbsvx)
extern void sgbsvx(
    char   *fact,
    char   *trans,
    ptrdiff_t *n,
    ptrdiff_t *kl,
    ptrdiff_t *ku,
    ptrdiff_t *nrhs,
    float  *ab,
    ptrdiff_t *ldab,
    float  *afb,
    ptrdiff_t *ldafb,
    ptrdiff_t *ipiv,
    char   *equed,
    float  *r,
    float  *c,
    float  *b,
    ptrdiff_t *ldb,
    float  *x,
    ptrdiff_t *ldx,
    float  *rcond,
    float  *ferr,
    float  *berr,
    float  *work,
    ptrdiff_t *iwork,
    ptrdiff_t *info
);

/* Source: sgbtf2.f */
#define sgbtf2 FORTRAN_WRAPPER(sgbtf2)
extern void sgbtf2(
    ptrdiff_t *m,
    ptrdiff_t *n,
    ptrdiff_t *kl,
    ptrdiff_t *ku,
    float  *ab,
    ptrdiff_t *ldab,
    ptrdiff_t *ipiv,
    ptrdiff_t *info
);

/* Source: sgbtrf.f */
#define sgbtrf FORTRAN_WRAPPER(sgbtrf)
extern void sgbtrf(
    ptrdiff_t *m,
    ptrdiff_t *n,
    ptrdiff_t *kl,
    ptrdiff_t *ku,
    float  *ab,
    ptrdiff_t *ldab,
    ptrdiff_t *ipiv,
    ptrdiff_t *info
);

/* Source: sgbtrs.f */
#define sgbtrs FORTRAN_WRAPPER(sgbtrs)
extern void sgbtrs(
    char   *trans,
    ptrdiff_t *n,
    ptrdiff_t *kl,
    ptrdiff_t *ku,
    ptrdiff_t *nrhs,
    float  *ab,
    ptrdiff_t *ldab,
    ptrdiff_t *ipiv,
    float  *b,
    ptrdiff_t *ldb,
    ptrdiff_t *info
);

/* Source: sgebak.f */
#define sgebak FORTRAN_WRAPPER(sgebak)
extern void sgebak(
    char   *job,
    char   *side,
    ptrdiff_t *n,
    ptrdiff_t *ilo,
    ptrdiff_t *ihi,
    float  *scale,
    ptrdiff_t *m,
    float  *v,
    ptrdiff_t *ldv,
    ptrdiff_t *info
);

/* Source: sgebal.f */
#define sgebal FORTRAN_WRAPPER(sgebal)
extern void sgebal(
    char   *job,
    ptrdiff_t *n,
    float  *a,
    ptrdiff_t *lda,
    ptrdiff_t *ilo,
    ptrdiff_t *ihi,
    float  *scale,
    ptrdiff_t *info
);

/* Source: sgebd2.f */
#define sgebd2 FORTRAN_WRAPPER(sgebd2)
extern void sgebd2(
    ptrdiff_t *m,
    ptrdiff_t *n,
    float  *a,
    ptrdiff_t *lda,
    float  *d,
    float  *e,
    float  *tauq,
    float  *taup,
    float  *work,
    ptrdiff_t *info
);

/* Source: sgebrd.f */
#define sgebrd FORTRAN_WRAPPER(sgebrd)
extern void sgebrd(
    ptrdiff_t *m,
    ptrdiff_t *n,
    float  *a,
    ptrdiff_t *lda,
    float  *d,
    float  *e,
    float  *tauq,
    float  *taup,
    float  *work,
    ptrdiff_t *lwork,
    ptrdiff_t *info
);

/* Source: sgecon.f */
#define sgecon FORTRAN_WRAPPER(sgecon)
extern void sgecon(
    char   *norm,
    ptrdiff_t *n,
    float  *a,
    ptrdiff_t *lda,
    float  *anorm,
    float  *rcond,
    float  *work,
    ptrdiff_t *iwork,
    ptrdiff_t *info
);

/* Source: sgeequ.f */
#define sgeequ FORTRAN_WRAPPER(sgeequ)
extern void sgeequ(
    ptrdiff_t *m,
    ptrdiff_t *n,
    float  *a,
    ptrdiff_t *lda,
    float  *r,
    float  *c,
    float  *rowcnd,
    float  *colcnd,
    float  *amax,
    ptrdiff_t *info
);

/* Source: sgeequb.f */
#define sgeequb FORTRAN_WRAPPER(sgeequb)
extern void sgeequb(
    ptrdiff_t *m,
    ptrdiff_t *n,
    float  *a,
    ptrdiff_t *lda,
    float  *r,
    float  *c,
    float  *rowcnd,
    float  *colcnd,
    float  *amax,
    ptrdiff_t *info
);

/* Source: sgees.f */
#define sgees FORTRAN_WRAPPER(sgees)
extern void sgees(
    char   *jobvs,
    char   *sort,
    ptrdiff_t (*select)(),
    ptrdiff_t *n,
    float  *a,
    ptrdiff_t *lda,
    ptrdiff_t *sdim,
    float  *wr,
    float  *wi,
    float  *vs,
    ptrdiff_t *ldvs,
    float  *work,
    ptrdiff_t *lwork,
    ptrdiff_t *bwork,
    ptrdiff_t *info
);

/* Source: sgeesx.f */
#define sgeesx FORTRAN_WRAPPER(sgeesx)
extern void sgeesx(
    char   *jobvs,
    char   *sort,
    ptrdiff_t (*select)(),
    char   *sense,
    ptrdiff_t *n,
    float  *a,
    ptrdiff_t *lda,
    ptrdiff_t *sdim,
    float  *wr,
    float  *wi,
    float  *vs,
    ptrdiff_t *ldvs,
    float  *rconde,
    float  *rcondv,
    float  *work,
    ptrdiff_t *lwork,
    ptrdiff_t *iwork,
    ptrdiff_t *liwork,
    ptrdiff_t *bwork,
    ptrdiff_t *info
);

/* Source: sgeev.f */
#define sgeev FORTRAN_WRAPPER(sgeev)
extern void sgeev(
    char   *jobvl,
    char   *jobvr,
    ptrdiff_t *n,
    float  *a,
    ptrdiff_t *lda,
    float  *wr,
    float  *wi,
    float  *vl,
    ptrdiff_t *ldvl,
    float  *vr,
    ptrdiff_t *ldvr,
    float  *work,
    ptrdiff_t *lwork,
    ptrdiff_t *info
);

/* Source: sgeevx.f */
#define sgeevx FORTRAN_WRAPPER(sgeevx)
extern void sgeevx(
    char   *balanc,
    char   *jobvl,
    char   *jobvr,
    char   *sense,
    ptrdiff_t *n,
    float  *a,
    ptrdiff_t *lda,
    float  *wr,
    float  *wi,
    float  *vl,
    ptrdiff_t *ldvl,
    float  *vr,
    ptrdiff_t *ldvr,
    ptrdiff_t *ilo,
    ptrdiff_t *ihi,
    float  *scale,
    float  *abnrm,
    float  *rconde,
    float  *rcondv,
    float  *work,
    ptrdiff_t *lwork,
    ptrdiff_t *iwork,
    ptrdiff_t *info
);

/* Source: sgegs.f */
#define sgegs FORTRAN_WRAPPER(sgegs)
extern void sgegs(
    char   *jobvsl,
    char   *jobvsr,
    ptrdiff_t *n,
    float  *a,
    ptrdiff_t *lda,
    float  *b,
    ptrdiff_t *ldb,
    float  *alphar,
    float  *alphai,
    float  *beta,
    float  *vsl,
    ptrdiff_t *ldvsl,
    float  *vsr,
    ptrdiff_t *ldvsr,
    float  *work,
    ptrdiff_t *lwork,
    ptrdiff_t *info
);

/* Source: sgegv.f */
#define sgegv FORTRAN_WRAPPER(sgegv)
extern void sgegv(
    char   *jobvl,
    char   *jobvr,
    ptrdiff_t *n,
    float  *a,
    ptrdiff_t *lda,
    float  *b,
    ptrdiff_t *ldb,
    float  *alphar,
    float  *alphai,
    float  *beta,
    float  *vl,
    ptrdiff_t *ldvl,
    float  *vr,
    ptrdiff_t *ldvr,
    float  *work,
    ptrdiff_t *lwork,
    ptrdiff_t *info
);

/* Source: sgehd2.f */
#define sgehd2 FORTRAN_WRAPPER(sgehd2)
extern void sgehd2(
    ptrdiff_t *n,
    ptrdiff_t *ilo,
    ptrdiff_t *ihi,
    float  *a,
    ptrdiff_t *lda,
    float  *tau,
    float  *work,
    ptrdiff_t *info
);

/* Source: sgehrd.f */
#define sgehrd FORTRAN_WRAPPER(sgehrd)
extern void sgehrd(
    ptrdiff_t *n,
    ptrdiff_t *ilo,
    ptrdiff_t *ihi,
    float  *a,
    ptrdiff_t *lda,
    float  *tau,
    float  *work,
    ptrdiff_t *lwork,
    ptrdiff_t *info
);

/* Source: sgejsv.f */
#define sgejsv FORTRAN_WRAPPER(sgejsv)
extern void sgejsv(
    char   *joba,
    char   *jobu,
    char   *jobv,
    char   *jobr,
    char   *jobt,
    char   *jobp,
    ptrdiff_t *m,
    ptrdiff_t *n,
    float  *a,
    ptrdiff_t *lda,
    float  *sva,
    float  *u,
    ptrdiff_t *ldu,
    float  *v,
    ptrdiff_t *ldv,
    float  *work,
    ptrdiff_t *lwork,
    ptrdiff_t *iwork,
    ptrdiff_t *info
);

/* Source: sgelq2.f */
#define sgelq2 FORTRAN_WRAPPER(sgelq2)
extern void sgelq2(
    ptrdiff_t *m,
    ptrdiff_t *n,
    float  *a,
    ptrdiff_t *lda,
    float  *tau,
    float  *work,
    ptrdiff_t *info
);

/* Source: sgelqf.f */
#define sgelqf FORTRAN_WRAPPER(sgelqf)
extern void sgelqf(
    ptrdiff_t *m,
    ptrdiff_t *n,
    float  *a,
    ptrdiff_t *lda,
    float  *tau,
    float  *work,
    ptrdiff_t *lwork,
    ptrdiff_t *info
);

/* Source: sgels.f */
#define sgels FORTRAN_WRAPPER(sgels)
extern void sgels(
    char   *trans,
    ptrdiff_t *m,
    ptrdiff_t *n,
    ptrdiff_t *nrhs,
    float  *a,
    ptrdiff_t *lda,
    float  *b,
    ptrdiff_t *ldb,
    float  *work,
    ptrdiff_t *lwork,
    ptrdiff_t *info
);

/* Source: sgelsd.f */
#define sgelsd FORTRAN_WRAPPER(sgelsd)
extern void sgelsd(
    ptrdiff_t *m,
    ptrdiff_t *n,
    ptrdiff_t *nrhs,
    float  *a,
    ptrdiff_t *lda,
    float  *b,
    ptrdiff_t *ldb,
    float  *s,
    float  *rcond,
    ptrdiff_t *rank,
    float  *work,
    ptrdiff_t *lwork,
    ptrdiff_t *iwork,
    ptrdiff_t *info
);

/* Source: sgelss.f */
#define sgelss FORTRAN_WRAPPER(sgelss)
extern void sgelss(
    ptrdiff_t *m,
    ptrdiff_t *n,
    ptrdiff_t *nrhs,
    float  *a,
    ptrdiff_t *lda,
    float  *b,
    ptrdiff_t *ldb,
    float  *s,
    float  *rcond,
    ptrdiff_t *rank,
    float  *work,
    ptrdiff_t *lwork,
    ptrdiff_t *info
);

/* Source: sgelsx.f */
#define sgelsx FORTRAN_WRAPPER(sgelsx)
extern void sgelsx(
    ptrdiff_t *m,
    ptrdiff_t *n,
    ptrdiff_t *nrhs,
    float  *a,
    ptrdiff_t *lda,
    float  *b,
    ptrdiff_t *ldb,
    ptrdiff_t *jpvt,
    float  *rcond,
    ptrdiff_t *rank,
    float  *work,
    ptrdiff_t *info
);

/* Source: sgelsy.f */
#define sgelsy FORTRAN_WRAPPER(sgelsy)
extern void sgelsy(
    ptrdiff_t *m,
    ptrdiff_t *n,
    ptrdiff_t *nrhs,
    float  *a,
    ptrdiff_t *lda,
    float  *b,
    ptrdiff_t *ldb,
    ptrdiff_t *jpvt,
    float  *rcond,
    ptrdiff_t *rank,
    float  *work,
    ptrdiff_t *lwork,
    ptrdiff_t *info
);

/* Source: sgeql2.f */
#define sgeql2 FORTRAN_WRAPPER(sgeql2)
extern void sgeql2(
    ptrdiff_t *m,
    ptrdiff_t *n,
    float  *a,
    ptrdiff_t *lda,
    float  *tau,
    float  *work,
    ptrdiff_t *info
);

/* Source: sgeqlf.f */
#define sgeqlf FORTRAN_WRAPPER(sgeqlf)
extern void sgeqlf(
    ptrdiff_t *m,
    ptrdiff_t *n,
    float  *a,
    ptrdiff_t *lda,
    float  *tau,
    float  *work,
    ptrdiff_t *lwork,
    ptrdiff_t *info
);

/* Source: sgeqp3.f */
#define sgeqp3 FORTRAN_WRAPPER(sgeqp3)
extern void sgeqp3(
    ptrdiff_t *m,
    ptrdiff_t *n,
    float  *a,
    ptrdiff_t *lda,
    ptrdiff_t *jpvt,
    float  *tau,
    float  *work,
    ptrdiff_t *lwork,
    ptrdiff_t *info
);

/* Source: sgeqpf.f */
#define sgeqpf FORTRAN_WRAPPER(sgeqpf)
extern void sgeqpf(
    ptrdiff_t *m,
    ptrdiff_t *n,
    float  *a,
    ptrdiff_t *lda,
    ptrdiff_t *jpvt,
    float  *tau,
    float  *work,
    ptrdiff_t *info
);

/* Source: sgeqr2.f */
#define sgeqr2 FORTRAN_WRAPPER(sgeqr2)
extern void sgeqr2(
    ptrdiff_t *m,
    ptrdiff_t *n,
    float  *a,
    ptrdiff_t *lda,
    float  *tau,
    float  *work,
    ptrdiff_t *info
);

/* Source: sgeqr2p.f */
#define sgeqr2p FORTRAN_WRAPPER(sgeqr2p)
extern void sgeqr2p(
    ptrdiff_t *m,
    ptrdiff_t *n,
    float  *a,
    ptrdiff_t *lda,
    float  *tau,
    float  *work,
    ptrdiff_t *info
);

/* Source: sgeqrf.f */
#define sgeqrf FORTRAN_WRAPPER(sgeqrf)
extern void sgeqrf(
    ptrdiff_t *m,
    ptrdiff_t *n,
    float  *a,
    ptrdiff_t *lda,
    float  *tau,
    float  *work,
    ptrdiff_t *lwork,
    ptrdiff_t *info
);

/* Source: sgeqrfp.f */
#define sgeqrfp FORTRAN_WRAPPER(sgeqrfp)
extern void sgeqrfp(
    ptrdiff_t *m,
    ptrdiff_t *n,
    float  *a,
    ptrdiff_t *lda,
    float  *tau,
    float  *work,
    ptrdiff_t *lwork,
    ptrdiff_t *info
);

/* Source: sgerfs.f */
#define sgerfs FORTRAN_WRAPPER(sgerfs)
extern void sgerfs(
    char   *trans,
    ptrdiff_t *n,
    ptrdiff_t *nrhs,
    float  *a,
    ptrdiff_t *lda,
    float  *af,
    ptrdiff_t *ldaf,
    ptrdiff_t *ipiv,
    float  *b,
    ptrdiff_t *ldb,
    float  *x,
    ptrdiff_t *ldx,
    float  *ferr,
    float  *berr,
    float  *work,
    ptrdiff_t *iwork,
    ptrdiff_t *info
);

/* Source: sgerq2.f */
#define sgerq2 FORTRAN_WRAPPER(sgerq2)
extern void sgerq2(
    ptrdiff_t *m,
    ptrdiff_t *n,
    float  *a,
    ptrdiff_t *lda,
    float  *tau,
    float  *work,
    ptrdiff_t *info
);

/* Source: sgerqf.f */
#define sgerqf FORTRAN_WRAPPER(sgerqf)
extern void sgerqf(
    ptrdiff_t *m,
    ptrdiff_t *n,
    float  *a,
    ptrdiff_t *lda,
    float  *tau,
    float  *work,
    ptrdiff_t *lwork,
    ptrdiff_t *info
);

/* Source: sgesc2.f */
#define sgesc2 FORTRAN_WRAPPER(sgesc2)
extern void sgesc2(
    ptrdiff_t *n,
    float  *a,
    ptrdiff_t *lda,
    float  *rhs,
    ptrdiff_t *ipiv,
    ptrdiff_t *jpiv,
    float  *scale
);

/* Source: sgesdd.f */
#define sgesdd FORTRAN_WRAPPER(sgesdd)
extern void sgesdd(
    char   *jobz,
    ptrdiff_t *m,
    ptrdiff_t *n,
    float  *a,
    ptrdiff_t *lda,
    float  *s,
    float  *u,
    ptrdiff_t *ldu,
    float  *vt,
    ptrdiff_t *ldvt,
    float  *work,
    ptrdiff_t *lwork,
    ptrdiff_t *iwork,
    ptrdiff_t *info
);

/* Source: sgesv.f */
#define sgesv FORTRAN_WRAPPER(sgesv)
extern void sgesv(
    ptrdiff_t *n,
    ptrdiff_t *nrhs,
    float  *a,
    ptrdiff_t *lda,
    ptrdiff_t *ipiv,
    float  *b,
    ptrdiff_t *ldb,
    ptrdiff_t *info
);

/* Source: sgesvd.f */
#define sgesvd FORTRAN_WRAPPER(sgesvd)
extern void sgesvd(
    char   *jobu,
    char   *jobvt,
    ptrdiff_t *m,
    ptrdiff_t *n,
    float  *a,
    ptrdiff_t *lda,
    float  *s,
    float  *u,
    ptrdiff_t *ldu,
    float  *vt,
    ptrdiff_t *ldvt,
    float  *work,
    ptrdiff_t *lwork,
    ptrdiff_t *info
);

/* Source: sgesvj.f */
#define sgesvj FORTRAN_WRAPPER(sgesvj)
extern void sgesvj(
    char   *joba,
    char   *jobu,
    char   *jobv,
    ptrdiff_t *m,
    ptrdiff_t *n,
    float  *a,
    ptrdiff_t *lda,
    float  *sva,
    ptrdiff_t *mv,
    float  *v,
    ptrdiff_t *ldv,
    float  *work,
    ptrdiff_t *lwork,
    ptrdiff_t *info
);

/* Source: sgesvx.f */
#define sgesvx FORTRAN_WRAPPER(sgesvx)
extern void sgesvx(
    char   *fact,
    char   *trans,
    ptrdiff_t *n,
    ptrdiff_t *nrhs,
    float  *a,
    ptrdiff_t *lda,
    float  *af,
    ptrdiff_t *ldaf,
    ptrdiff_t *ipiv,
    char   *equed,
    float  *r,
    float  *c,
    float  *b,
    ptrdiff_t *ldb,
    float  *x,
    ptrdiff_t *ldx,
    float  *rcond,
    float  *ferr,
    float  *berr,
    float  *work,
    ptrdiff_t *iwork,
    ptrdiff_t *info
);

/* Source: sgetc2.f */
#define sgetc2 FORTRAN_WRAPPER(sgetc2)
extern void sgetc2(
    ptrdiff_t *n,
    float  *a,
    ptrdiff_t *lda,
    ptrdiff_t *ipiv,
    ptrdiff_t *jpiv,
    ptrdiff_t *info
);

/* Source: sgetf2.f */
#define sgetf2 FORTRAN_WRAPPER(sgetf2)
extern void sgetf2(
    ptrdiff_t *m,
    ptrdiff_t *n,
    float  *a,
    ptrdiff_t *lda,
    ptrdiff_t *ipiv,
    ptrdiff_t *info
);

/* Source: sgetrf.f */
#define sgetrf FORTRAN_WRAPPER(sgetrf)
extern void sgetrf(
    ptrdiff_t *m,
    ptrdiff_t *n,
    float  *a,
    ptrdiff_t *lda,
    ptrdiff_t *ipiv,
    ptrdiff_t *info
);

/* Source: sgetri.f */
#define sgetri FORTRAN_WRAPPER(sgetri)
extern void sgetri(
    ptrdiff_t *n,
    float  *a,
    ptrdiff_t *lda,
    ptrdiff_t *ipiv,
    float  *work,
    ptrdiff_t *lwork,
    ptrdiff_t *info
);

/* Source: sgetrs.f */
#define sgetrs FORTRAN_WRAPPER(sgetrs)
extern void sgetrs(
    char   *trans,
    ptrdiff_t *n,
    ptrdiff_t *nrhs,
    float  *a,
    ptrdiff_t *lda,
    ptrdiff_t *ipiv,
    float  *b,
    ptrdiff_t *ldb,
    ptrdiff_t *info
);

/* Source: sggbak.f */
#define sggbak FORTRAN_WRAPPER(sggbak)
extern void sggbak(
    char   *job,
    char   *side,
    ptrdiff_t *n,
    ptrdiff_t *ilo,
    ptrdiff_t *ihi,
    float  *lscale,
    float  *rscale,
    ptrdiff_t *m,
    float  *v,
    ptrdiff_t *ldv,
    ptrdiff_t *info
);

/* Source: sggbal.f */
#define sggbal FORTRAN_WRAPPER(sggbal)
extern void sggbal(
    char   *job,
    ptrdiff_t *n,
    float  *a,
    ptrdiff_t *lda,
    float  *b,
    ptrdiff_t *ldb,
    ptrdiff_t *ilo,
    ptrdiff_t *ihi,
    float  *lscale,
    float  *rscale,
    float  *work,
    ptrdiff_t *info
);

/* Source: sgges.f */
#define sgges FORTRAN_WRAPPER(sgges)
extern void sgges(
    char   *jobvsl,
    char   *jobvsr,
    char   *sort,
    ptrdiff_t (*selctg)(),
    ptrdiff_t *n,
    float  *a,
    ptrdiff_t *lda,
    float  *b,
    ptrdiff_t *ldb,
    ptrdiff_t *sdim,
    float  *alphar,
    float  *alphai,
    float  *beta,
    float  *vsl,
    ptrdiff_t *ldvsl,
    float  *vsr,
    ptrdiff_t *ldvsr,
    float  *work,
    ptrdiff_t *lwork,
    ptrdiff_t *bwork,
    ptrdiff_t *info
);

/* Source: sggesx.f */
#define sggesx FORTRAN_WRAPPER(sggesx)
extern void sggesx(
    char   *jobvsl,
    char   *jobvsr,
    char   *sort,
    ptrdiff_t (*selctg)(),
    char   *sense,
    ptrdiff_t *n,
    float  *a,
    ptrdiff_t *lda,
    float  *b,
    ptrdiff_t *ldb,
    ptrdiff_t *sdim,
    float  *alphar,
    float  *alphai,
    float  *beta,
    float  *vsl,
    ptrdiff_t *ldvsl,
    float  *vsr,
    ptrdiff_t *ldvsr,
    float  *rconde,
    float  *rcondv,
    float  *work,
    ptrdiff_t *lwork,
    ptrdiff_t *iwork,
    ptrdiff_t *liwork,
    ptrdiff_t *bwork,
    ptrdiff_t *info
);

/* Source: sggev.f */
#define sggev FORTRAN_WRAPPER(sggev)
extern void sggev(
    char   *jobvl,
    char   *jobvr,
    ptrdiff_t *n,
    float  *a,
    ptrdiff_t *lda,
    float  *b,
    ptrdiff_t *ldb,
    float  *alphar,
    float  *alphai,
    float  *beta,
    float  *vl,
    ptrdiff_t *ldvl,
    float  *vr,
    ptrdiff_t *ldvr,
    float  *work,
    ptrdiff_t *lwork,
    ptrdiff_t *info
);

/* Source: sggevx.f */
#define sggevx FORTRAN_WRAPPER(sggevx)
extern void sggevx(
    char   *balanc,
    char   *jobvl,
    char   *jobvr,
    char   *sense,
    ptrdiff_t *n,
    float  *a,
    ptrdiff_t *lda,
    float  *b,
    ptrdiff_t *ldb,
    float  *alphar,
    float  *alphai,
    float  *beta,
    float  *vl,
    ptrdiff_t *ldvl,
    float  *vr,
    ptrdiff_t *ldvr,
    ptrdiff_t *ilo,
    ptrdiff_t *ihi,
    float  *lscale,
    float  *rscale,
    float  *abnrm,
    float  *bbnrm,
    float  *rconde,
    float  *rcondv,
    float  *work,
    ptrdiff_t *lwork,
    ptrdiff_t *iwork,
    ptrdiff_t *bwork,
    ptrdiff_t *info
);

/* Source: sggglm.f */
#define sggglm FORTRAN_WRAPPER(sggglm)
extern void sggglm(
    ptrdiff_t *n,
    ptrdiff_t *m,
    ptrdiff_t *p,
    float  *a,
    ptrdiff_t *lda,
    float  *b,
    ptrdiff_t *ldb,
    float  *d,
    float  *x,
    float  *y,
    float  *work,
    ptrdiff_t *lwork,
    ptrdiff_t *info
);

/* Source: sgghrd.f */
#define sgghrd FORTRAN_WRAPPER(sgghrd)
extern void sgghrd(
    char   *compq,
    char   *compz,
    ptrdiff_t *n,
    ptrdiff_t *ilo,
    ptrdiff_t *ihi,
    float  *a,
    ptrdiff_t *lda,
    float  *b,
    ptrdiff_t *ldb,
    float  *q,
    ptrdiff_t *ldq,
    float  *z,
    ptrdiff_t *ldz,
    ptrdiff_t *info
);

/* Source: sgglse.f */
#define sgglse FORTRAN_WRAPPER(sgglse)
extern void sgglse(
    ptrdiff_t *m,
    ptrdiff_t *n,
    ptrdiff_t *p,
    float  *a,
    ptrdiff_t *lda,
    float  *b,
    ptrdiff_t *ldb,
    float  *c,
    float  *d,
    float  *x,
    float  *work,
    ptrdiff_t *lwork,
    ptrdiff_t *info
);

/* Source: sggqrf.f */
#define sggqrf FORTRAN_WRAPPER(sggqrf)
extern void sggqrf(
    ptrdiff_t *n,
    ptrdiff_t *m,
    ptrdiff_t *p,
    float  *a,
    ptrdiff_t *lda,
    float  *taua,
    float  *b,
    ptrdiff_t *ldb,
    float  *taub,
    float  *work,
    ptrdiff_t *lwork,
    ptrdiff_t *info
);

/* Source: sggrqf.f */
#define sggrqf FORTRAN_WRAPPER(sggrqf)
extern void sggrqf(
    ptrdiff_t *m,
    ptrdiff_t *p,
    ptrdiff_t *n,
    float  *a,
    ptrdiff_t *lda,
    float  *taua,
    float  *b,
    ptrdiff_t *ldb,
    float  *taub,
    float  *work,
    ptrdiff_t *lwork,
    ptrdiff_t *info
);

/* Source: sggsvd.f */
#define sggsvd FORTRAN_WRAPPER(sggsvd)
extern void sggsvd(
    char   *jobu,
    char   *jobv,
    char   *jobq,
    ptrdiff_t *m,
    ptrdiff_t *n,
    ptrdiff_t *p,
    ptrdiff_t *k,
    ptrdiff_t *l,
    float  *a,
    ptrdiff_t *lda,
    float  *b,
    ptrdiff_t *ldb,
    float  *alpha,
    float  *beta,
    float  *u,
    ptrdiff_t *ldu,
    float  *v,
    ptrdiff_t *ldv,
    float  *q,
    ptrdiff_t *ldq,
    float  *work,
    ptrdiff_t *iwork,
    ptrdiff_t *info
);

/* Source: sggsvp.f */
#define sggsvp FORTRAN_WRAPPER(sggsvp)
extern void sggsvp(
    char   *jobu,
    char   *jobv,
    char   *jobq,
    ptrdiff_t *m,
    ptrdiff_t *p,
    ptrdiff_t *n,
    float  *a,
    ptrdiff_t *lda,
    float  *b,
    ptrdiff_t *ldb,
    float  *tola,
    float  *tolb,
    ptrdiff_t *k,
    ptrdiff_t *l,
    float  *u,
    ptrdiff_t *ldu,
    float  *v,
    ptrdiff_t *ldv,
    float  *q,
    ptrdiff_t *ldq,
    ptrdiff_t *iwork,
    float  *tau,
    float  *work,
    ptrdiff_t *info
);

/* Source: sgsvj0.f */
#define sgsvj0 FORTRAN_WRAPPER(sgsvj0)
extern void sgsvj0(
    char   *jobv,
    ptrdiff_t *m,
    ptrdiff_t *n,
    float  *a,
    ptrdiff_t *lda,
    float  *d,
    float  *sva,
    ptrdiff_t *mv,
    float  *v,
    ptrdiff_t *ldv,
    float  *eps,
    float  *sfmin,
    float  *tol,
    ptrdiff_t *nsweep,
    float  *work,
    ptrdiff_t *lwork,
    ptrdiff_t *info
);

/* Source: sgsvj1.f */
#define sgsvj1 FORTRAN_WRAPPER(sgsvj1)
extern void sgsvj1(
    char   *jobv,
    ptrdiff_t *m,
    ptrdiff_t *n,
    ptrdiff_t *n1,
    float  *a,
    ptrdiff_t *lda,
    float  *d,
    float  *sva,
    ptrdiff_t *mv,
    float  *v,
    ptrdiff_t *ldv,
    float  *eps,
    float  *sfmin,
    float  *tol,
    ptrdiff_t *nsweep,
    float  *work,
    ptrdiff_t *lwork,
    ptrdiff_t *info
);

/* Source: sgtcon.f */
#define sgtcon FORTRAN_WRAPPER(sgtcon)
extern void sgtcon(
    char   *norm,
    ptrdiff_t *n,
    float  *dl,
    float  *d,
    float  *du,
    float  *du2,
    ptrdiff_t *ipiv,
    float  *anorm,
    float  *rcond,
    float  *work,
    ptrdiff_t *iwork,
    ptrdiff_t *info
);

/* Source: sgtrfs.f */
#define sgtrfs FORTRAN_WRAPPER(sgtrfs)
extern void sgtrfs(
    char   *trans,
    ptrdiff_t *n,
    ptrdiff_t *nrhs,
    float  *dl,
    float  *d,
    float  *du,
    float  *dlf,
    float  *df,
    float  *duf,
    float  *du2,
    ptrdiff_t *ipiv,
    float  *b,
    ptrdiff_t *ldb,
    float  *x,
    ptrdiff_t *ldx,
    float  *ferr,
    float  *berr,
    float  *work,
    ptrdiff_t *iwork,
    ptrdiff_t *info
);

/* Source: sgtsv.f */
#define sgtsv FORTRAN_WRAPPER(sgtsv)
extern void sgtsv(
    ptrdiff_t *n,
    ptrdiff_t *nrhs,
    float  *dl,
    float  *d,
    float  *du,
    float  *b,
    ptrdiff_t *ldb,
    ptrdiff_t *info
);

/* Source: sgtsvx.f */
#define sgtsvx FORTRAN_WRAPPER(sgtsvx)
extern void sgtsvx(
    char   *fact,
    char   *trans,
    ptrdiff_t *n,
    ptrdiff_t *nrhs,
    float  *dl,
    float  *d,
    float  *du,
    float  *dlf,
    float  *df,
    float  *duf,
    float  *du2,
    ptrdiff_t *ipiv,
    float  *b,
    ptrdiff_t *ldb,
    float  *x,
    ptrdiff_t *ldx,
    float  *rcond,
    float  *ferr,
    float  *berr,
    float  *work,
    ptrdiff_t *iwork,
    ptrdiff_t *info
);

/* Source: sgttrf.f */
#define sgttrf FORTRAN_WRAPPER(sgttrf)
extern void sgttrf(
    ptrdiff_t *n,
    float  *dl,
    float  *d,
    float  *du,
    float  *du2,
    ptrdiff_t *ipiv,
    ptrdiff_t *info
);

/* Source: sgttrs.f */
#define sgttrs FORTRAN_WRAPPER(sgttrs)
extern void sgttrs(
    char   *trans,
    ptrdiff_t *n,
    ptrdiff_t *nrhs,
    float  *dl,
    float  *d,
    float  *du,
    float  *du2,
    ptrdiff_t *ipiv,
    float  *b,
    ptrdiff_t *ldb,
    ptrdiff_t *info
);

/* Source: sgtts2.f */
#define sgtts2 FORTRAN_WRAPPER(sgtts2)
extern void sgtts2(
    ptrdiff_t *itrans,
    ptrdiff_t *n,
    ptrdiff_t *nrhs,
    float  *dl,
    float  *d,
    float  *du,
    float  *du2,
    ptrdiff_t *ipiv,
    float  *b,
    ptrdiff_t *ldb
);

/* Source: shgeqz.f */
#define shgeqz FORTRAN_WRAPPER(shgeqz)
extern void shgeqz(
    char   *job,
    char   *compq,
    char   *compz,
    ptrdiff_t *n,
    ptrdiff_t *ilo,
    ptrdiff_t *ihi,
    float  *h,
    ptrdiff_t *ldh,
    float  *t,
    ptrdiff_t *ldt,
    float  *alphar,
    float  *alphai,
    float  *beta,
    float  *q,
    ptrdiff_t *ldq,
    float  *z,
    ptrdiff_t *ldz,
    float  *work,
    ptrdiff_t *lwork,
    ptrdiff_t *info
);

/* Source: shsein.f */
#define shsein FORTRAN_WRAPPER(shsein)
extern void shsein(
    char   *side,
    char   *eigsrc,
    char   *initv,
    ptrdiff_t *select,
    ptrdiff_t *n,
    float  *h,
    ptrdiff_t *ldh,
    float  *wr,
    float  *wi,
    float  *vl,
    ptrdiff_t *ldvl,
    float  *vr,
    ptrdiff_t *ldvr,
    ptrdiff_t *mm,
    ptrdiff_t *m,
    float  *work,
    ptrdiff_t *ifaill,
    ptrdiff_t *ifailr,
    ptrdiff_t *info
);

/* Source: shseqr.f */
#define shseqr FORTRAN_WRAPPER(shseqr)
extern void shseqr(
    char   *job,
    char   *compz,
    ptrdiff_t *n,
    ptrdiff_t *ilo,
    ptrdiff_t *ihi,
    float  *h,
    ptrdiff_t *ldh,
    float  *wr,
    float  *wi,
    float  *z,
    ptrdiff_t *ldz,
    float  *work,
    ptrdiff_t *lwork,
    ptrdiff_t *info
);

/* Source: sisnan.f */
#define sisnan FORTRAN_WRAPPER(sisnan)
extern ptrdiff_t sisnan(
    float  *sin
);

/* Source: slabad.f */
#define slabad FORTRAN_WRAPPER(slabad)
extern void slabad(
    float  *small,
    float  *large
);

/* Source: slabrd.f */
#define slabrd FORTRAN_WRAPPER(slabrd)
extern void slabrd(
    ptrdiff_t *m,
    ptrdiff_t *n,
    ptrdiff_t *nb,
    float  *a,
    ptrdiff_t *lda,
    float  *d,
    float  *e,
    float  *tauq,
    float  *taup,
    float  *x,
    ptrdiff_t *ldx,
    float  *y,
    ptrdiff_t *ldy
);

/* Source: slacn2.f */
#define slacn2 FORTRAN_WRAPPER(slacn2)
extern void slacn2(
    ptrdiff_t *n,
    float  *v,
    float  *x,
    ptrdiff_t *isgn,
    float  *est,
    ptrdiff_t *kase,
    ptrdiff_t *isave
);

/* Source: slacon.f */
#define slacon FORTRAN_WRAPPER(slacon)
extern void slacon(
    ptrdiff_t *n,
    float  *v,
    float  *x,
    ptrdiff_t *isgn,
    float  *est,
    ptrdiff_t *kase
);

/* Source: slacpy.f */
#define slacpy FORTRAN_WRAPPER(slacpy)
extern void slacpy(
    char   *uplo,
    ptrdiff_t *m,
    ptrdiff_t *n,
    float  *a,
    ptrdiff_t *lda,
    float  *b,
    ptrdiff_t *ldb
);

/* Source: sladiv.f */
#define sladiv FORTRAN_WRAPPER(sladiv)
extern void sladiv(
    float  *a,
    float  *b,
    float  *c,
    float  *d,
    float  *p,
    float  *q
);

/* Source: slae2.f */
#define slae2 FORTRAN_WRAPPER(slae2)
extern void slae2(
    float  *a,
    float  *b,
    float  *c,
    float  *rt1,
    float  *rt2
);

/* Source: slaebz.f */
#define slaebz FORTRAN_WRAPPER(slaebz)
extern void slaebz(
    ptrdiff_t *ijob,
    ptrdiff_t *nitmax,
    ptrdiff_t *n,
    ptrdiff_t *mmax,
    ptrdiff_t *minp,
    ptrdiff_t *nbmin,
    float  *abstol,
    float  *reltol,
    float  *pivmin,
    float  *d,
    float  *e,
    float  *e2,
    ptrdiff_t *nval,
    float  *ab,
    float  *c,
    ptrdiff_t *mout,
    ptrdiff_t *nab,
    float  *work,
    ptrdiff_t *iwork,
    ptrdiff_t *info
);

/* Source: slaed0.f */
#define slaed0 FORTRAN_WRAPPER(slaed0)
extern void slaed0(
    ptrdiff_t *icompq,
    ptrdiff_t *qsiz,
    ptrdiff_t *n,
    float  *d,
    float  *e,
    float  *q,
    ptrdiff_t *ldq,
    float  *qstore,
    ptrdiff_t *ldqs,
    float  *work,
    ptrdiff_t *iwork,
    ptrdiff_t *info
);

/* Source: slaed1.f */
#define slaed1 FORTRAN_WRAPPER(slaed1)
extern void slaed1(
    ptrdiff_t *n,
    float  *d,
    float  *q,
    ptrdiff_t *ldq,
    ptrdiff_t *indxq,
    float  *rho,
    ptrdiff_t *cutpnt,
    float  *work,
    ptrdiff_t *iwork,
    ptrdiff_t *info
);

/* Source: slaed2.f */
#define slaed2 FORTRAN_WRAPPER(slaed2)
extern void slaed2(
    ptrdiff_t *k,
    ptrdiff_t *n,
    ptrdiff_t *n1,
    float  *d,
    float  *q,
    ptrdiff_t *ldq,
    ptrdiff_t *indxq,
    float  *rho,
    float  *z,
    float  *dlamda,
    float  *w,
    float  *q2,
    ptrdiff_t *indx,
    ptrdiff_t *indxc,
    ptrdiff_t *indxp,
    ptrdiff_t *coltyp,
    ptrdiff_t *info
);

/* Source: slaed3.f */
#define slaed3 FORTRAN_WRAPPER(slaed3)
extern void slaed3(
    ptrdiff_t *k,
    ptrdiff_t *n,
    ptrdiff_t *n1,
    float  *d,
    float  *q,
    ptrdiff_t *ldq,
    float  *rho,
    float  *dlamda,
    float  *q2,
    ptrdiff_t *indx,
    ptrdiff_t *ctot,
    float  *w,
    float  *s,
    ptrdiff_t *info
);

/* Source: slaed4.f */
#define slaed4 FORTRAN_WRAPPER(slaed4)
extern void slaed4(
    ptrdiff_t *n,
    ptrdiff_t *i,
    float  *d,
    float  *z,
    float  *delta,
    float  *rho,
    float  *dlam,
    ptrdiff_t *info
);

/* Source: slaed5.f */
#define slaed5 FORTRAN_WRAPPER(slaed5)
extern void slaed5(
    ptrdiff_t *i,
    float  *d,
    float  *z,
    float  *delta,
    float  *rho,
    float  *dlam
);

/* Source: slaed6.f */
#define slaed6 FORTRAN_WRAPPER(slaed6)
extern void slaed6(
    ptrdiff_t *kniter,
    ptrdiff_t *orgati,
    float  *rho,
    float  *d,
    float  *z,
    float  *finit,
    float  *tau,
    ptrdiff_t *info
);

/* Source: slaed7.f */
#define slaed7 FORTRAN_WRAPPER(slaed7)
extern void slaed7(
    ptrdiff_t *icompq,
    ptrdiff_t *n,
    ptrdiff_t *qsiz,
    ptrdiff_t *tlvls,
    ptrdiff_t *curlvl,
    ptrdiff_t *curpbm,
    float  *d,
    float  *q,
    ptrdiff_t *ldq,
    ptrdiff_t *indxq,
    float  *rho,
    ptrdiff_t *cutpnt,
    float  *qstore,
    ptrdiff_t *qptr,
    ptrdiff_t *prmptr,
    ptrdiff_t *perm,
    ptrdiff_t *givptr,
    ptrdiff_t *givcol,
    float  *givnum,
    float  *work,
    ptrdiff_t *iwork,
    ptrdiff_t *info
);

/* Source: slaed8.f */
#define slaed8 FORTRAN_WRAPPER(slaed8)
extern void slaed8(
    ptrdiff_t *icompq,
    ptrdiff_t *k,
    ptrdiff_t *n,
    ptrdiff_t *qsiz,
    float  *d,
    float  *q,
    ptrdiff_t *ldq,
    ptrdiff_t *indxq,
    float  *rho,
    ptrdiff_t *cutpnt,
    float  *z,
    float  *dlamda,
    float  *q2,
    ptrdiff_t *ldq2,
    float  *w,
    ptrdiff_t *perm,
    ptrdiff_t *givptr,
    ptrdiff_t *givcol,
    float  *givnum,
    ptrdiff_t *indxp,
    ptrdiff_t *indx,
    ptrdiff_t *info
);

/* Source: slaed9.f */
#define slaed9 FORTRAN_WRAPPER(slaed9)
extern void slaed9(
    ptrdiff_t *k,
    ptrdiff_t *kstart,
    ptrdiff_t *kstop,
    ptrdiff_t *n,
    float  *d,
    float  *q,
    ptrdiff_t *ldq,
    float  *rho,
    float  *dlamda,
    float  *w,
    float  *s,
    ptrdiff_t *lds,
    ptrdiff_t *info
);

/* Source: slaeda.f */
#define slaeda FORTRAN_WRAPPER(slaeda)
extern void slaeda(
    ptrdiff_t *n,
    ptrdiff_t *tlvls,
    ptrdiff_t *curlvl,
    ptrdiff_t *curpbm,
    ptrdiff_t *prmptr,
    ptrdiff_t *perm,
    ptrdiff_t *givptr,
    ptrdiff_t *givcol,
    float  *givnum,
    float  *q,
    ptrdiff_t *qptr,
    float  *z,
    float  *ztemp,
    ptrdiff_t *info
);

/* Source: slaein.f */
#define slaein FORTRAN_WRAPPER(slaein)
extern void slaein(
    ptrdiff_t *rightv,
    ptrdiff_t *noinit,
    ptrdiff_t *n,
    float  *h,
    ptrdiff_t *ldh,
    float  *wr,
    float  *wi,
    float  *vr,
    float  *vi,
    float  *b,
    ptrdiff_t *ldb,
    float  *work,
    float  *eps3,
    float  *smlnum,
    float  *bignum,
    ptrdiff_t *info
);

/* Source: slaev2.f */
#define slaev2 FORTRAN_WRAPPER(slaev2)
extern void slaev2(
    float  *a,
    float  *b,
    float  *c,
    float  *rt1,
    float  *rt2,
    float  *cs1,
    float  *sn1
);

/* Source: slaexc.f */
#define slaexc FORTRAN_WRAPPER(slaexc)
extern void slaexc(
    ptrdiff_t *wantq,
    ptrdiff_t *n,
    float  *t,
    ptrdiff_t *ldt,
    float  *q,
    ptrdiff_t *ldq,
    ptrdiff_t *j1_,
    ptrdiff_t *n1,
    ptrdiff_t *n2,
    float  *work,
    ptrdiff_t *info
);

/* Source: slag2.f */
#define slag2 FORTRAN_WRAPPER(slag2)
extern void slag2(
    float  *a,
    ptrdiff_t *lda,
    float  *b,
    ptrdiff_t *ldb,
    float  *safmin,
    float  *scale1,
    float  *scale2,
    float  *wr1,
    float  *wr2,
    float  *wi
);

/* Source: slag2d.f */
#define slag2d FORTRAN_WRAPPER(slag2d)
extern void slag2d(
    ptrdiff_t *m,
    ptrdiff_t *n,
    float  *sa,
    ptrdiff_t *ldsa,
    double *a,
    ptrdiff_t *lda,
    ptrdiff_t *info
);

/* Source: slags2.f */
#define slags2 FORTRAN_WRAPPER(slags2)
extern void slags2(
    ptrdiff_t *upper,
    float  *a1,
    float  *a2,
    float  *a3,
    float  *b1,
    float  *b2,
    float  *b3,
    float  *csu,
    float  *snu,
    float  *csv,
    float  *snv,
    float  *csq,
    float  *snq
);

/* Source: slagtf.f */
#define slagtf FORTRAN_WRAPPER(slagtf)
extern void slagtf(
    ptrdiff_t *n,
    float  *a,
    float  *lambda,
    float  *b,
    float  *c,
    float  *tol,
    float  *d,
    ptrdiff_t *in,
    ptrdiff_t *info
);

/* Source: slagtm.f */
#define slagtm FORTRAN_WRAPPER(slagtm)
extern void slagtm(
    char   *trans,
    ptrdiff_t *n,
    ptrdiff_t *nrhs,
    float  *alpha,
    float  *dl,
    float  *d,
    float  *du,
    float  *x,
    ptrdiff_t *ldx,
    float  *beta,
    float  *b,
    ptrdiff_t *ldb
);

/* Source: slagts.f */
#define slagts FORTRAN_WRAPPER(slagts)
extern void slagts(
    ptrdiff_t *job,
    ptrdiff_t *n,
    float  *a,
    float  *b,
    float  *c,
    float  *d,
    ptrdiff_t *in,
    float  *y,
    float  *tol,
    ptrdiff_t *info
);

/* Source: slagv2.f */
#define slagv2 FORTRAN_WRAPPER(slagv2)
extern void slagv2(
    float  *a,
    ptrdiff_t *lda,
    float  *b,
    ptrdiff_t *ldb,
    float  *alphar,
    float  *alphai,
    float  *beta,
    float  *csl,
    float  *snl,
    float  *csr,
    float  *snr
);

/* Source: slahqr.f */
#define slahqr FORTRAN_WRAPPER(slahqr)
extern void slahqr(
    ptrdiff_t *wantt,
    ptrdiff_t *wantz,
    ptrdiff_t *n,
    ptrdiff_t *ilo,
    ptrdiff_t *ihi,
    float  *h,
    ptrdiff_t *ldh,
    float  *wr,
    float  *wi,
    ptrdiff_t *iloz,
    ptrdiff_t *ihiz,
    float  *z,
    ptrdiff_t *ldz,
    ptrdiff_t *info
);

/* Source: slahr2.f */
#define slahr2 FORTRAN_WRAPPER(slahr2)
extern void slahr2(
    ptrdiff_t *n,
    ptrdiff_t *k,
    ptrdiff_t *nb,
    float  *a,
    ptrdiff_t *lda,
    float  *tau,
    float  *t,
    ptrdiff_t *ldt,
    float  *y,
    ptrdiff_t *ldy
);

/* Source: slahrd.f */
#define slahrd FORTRAN_WRAPPER(slahrd)
extern void slahrd(
    ptrdiff_t *n,
    ptrdiff_t *k,
    ptrdiff_t *nb,
    float  *a,
    ptrdiff_t *lda,
    float  *tau,
    float  *t,
    ptrdiff_t *ldt,
    float  *y,
    ptrdiff_t *ldy
);

/* Source: slaic1.f */
#define slaic1 FORTRAN_WRAPPER(slaic1)
extern void slaic1(
    ptrdiff_t *job,
    ptrdiff_t *j,
    float  *x,
    float  *sest,
    float  *w,
    float  *gamma_,
    float  *sestpr,
    float  *s,
    float  *c
);

/* Source: slaisnan.f */
#define slaisnan FORTRAN_WRAPPER(slaisnan)
extern ptrdiff_t slaisnan(
    float  *sin1,
    float  *sin2
);

/* Source: slaln2.f */
#define slaln2 FORTRAN_WRAPPER(slaln2)
extern void slaln2(
    ptrdiff_t *ltrans,
    ptrdiff_t *na,
    ptrdiff_t *nw,
    float  *smin,
    float  *ca,
    float  *a,
    ptrdiff_t *lda,
    float  *d1,
    float  *d2,
    float  *b,
    ptrdiff_t *ldb,
    float  *wr,
    float  *wi,
    float  *x,
    ptrdiff_t *ldx,
    float  *scale,
    float  *xnorm,
    ptrdiff_t *info
);

/* Source: slals0.f */
#define slals0 FORTRAN_WRAPPER(slals0)
extern void slals0(
    ptrdiff_t *icompq,
    ptrdiff_t *nl,
    ptrdiff_t *nr,
    ptrdiff_t *sqre,
    ptrdiff_t *nrhs,
    float  *b,
    ptrdiff_t *ldb,
    float  *bx,
    ptrdiff_t *ldbx,
    ptrdiff_t *perm,
    ptrdiff_t *givptr,
    ptrdiff_t *givcol,
    ptrdiff_t *ldgcol,
    float  *givnum,
    ptrdiff_t *ldgnum,
    float  *poles,
    float  *difl,
    float  *difr,
    float  *z,
    ptrdiff_t *k,
    float  *c,
    float  *s,
    float  *work,
    ptrdiff_t *info
);

/* Source: slalsa.f */
#define slalsa FORTRAN_WRAPPER(slalsa)
extern void slalsa(
    ptrdiff_t *icompq,
    ptrdiff_t *smlsiz,
    ptrdiff_t *n,
    ptrdiff_t *nrhs,
    float  *b,
    ptrdiff_t *ldb,
    float  *bx,
    ptrdiff_t *ldbx,
    float  *u,
    ptrdiff_t *ldu,
    float  *vt,
    ptrdiff_t *k,
    float  *difl,
    float  *difr,
    float  *z,
    float  *poles,
    ptrdiff_t *givptr,
    ptrdiff_t *givcol,
    ptrdiff_t *ldgcol,
    ptrdiff_t *perm,
    float  *givnum,
    float  *c,
    float  *s,
    float  *work,
    ptrdiff_t *iwork,
    ptrdiff_t *info
);

/* Source: slalsd.f */
#define slalsd FORTRAN_WRAPPER(slalsd)
extern void slalsd(
    char   *uplo,
    ptrdiff_t *smlsiz,
    ptrdiff_t *n,
    ptrdiff_t *nrhs,
    float  *d,
    float  *e,
    float  *b,
    ptrdiff_t *ldb,
    float  *rcond,
    ptrdiff_t *rank,
    float  *work,
    ptrdiff_t *iwork,
    ptrdiff_t *info
);

/* Source: slamrg.f */
#define slamrg FORTRAN_WRAPPER(slamrg)
extern void slamrg(
    ptrdiff_t *n1,
    ptrdiff_t *n2,
    float  *a,
    ptrdiff_t *strd1,
    ptrdiff_t *strd2,
    ptrdiff_t *index
);

/* Source: slaneg.f */
#define slaneg FORTRAN_WRAPPER(slaneg)
extern ptrdiff_t slaneg(
    ptrdiff_t *n,
    float  *d,
    float  *lld,
    float  *sigma,
    float  *pivmin,
    ptrdiff_t *r
);

/* Source: slangb.f */
#define slangb FORTRAN_WRAPPER(slangb)
#ifdef FORTRAN_FLOAT_FUNCTIONS_RETURN_DOUBLE
extern double slangb(
#else
extern float slangb(
#endif
    char   *norm,
    ptrdiff_t *n,
    ptrdiff_t *kl,
    ptrdiff_t *ku,
    float  *ab,
    ptrdiff_t *ldab,
    float  *work
);

/* Source: slange.f */
#define slange FORTRAN_WRAPPER(slange)
#ifdef FORTRAN_FLOAT_FUNCTIONS_RETURN_DOUBLE
extern double slange(
#else
extern float slange(
#endif
    char   *norm,
    ptrdiff_t *m,
    ptrdiff_t *n,
    float  *a,
    ptrdiff_t *lda,
    float  *work
);

/* Source: slangt.f */
#define slangt FORTRAN_WRAPPER(slangt)
#ifdef FORTRAN_FLOAT_FUNCTIONS_RETURN_DOUBLE
extern double slangt(
#else
extern float slangt(
#endif
    char   *norm,
    ptrdiff_t *n,
    float  *dl,
    float  *d,
    float  *du
);

/* Source: slanhs.f */
#define slanhs FORTRAN_WRAPPER(slanhs)
#ifdef FORTRAN_FLOAT_FUNCTIONS_RETURN_DOUBLE
extern double slanhs(
#else
extern float slanhs(
#endif
    char   *norm,
    ptrdiff_t *n,
    float  *a,
    ptrdiff_t *lda,
    float  *work
);

/* Source: slansb.f */
#define slansb FORTRAN_WRAPPER(slansb)
#ifdef FORTRAN_FLOAT_FUNCTIONS_RETURN_DOUBLE
extern double slansb(
#else
extern float slansb(
#endif
    char   *norm,
    char   *uplo,
    ptrdiff_t *n,
    ptrdiff_t *k,
    float  *ab,
    ptrdiff_t *ldab,
    float  *work
);

/* Source: slansf.f */
#define slansf FORTRAN_WRAPPER(slansf)
#ifdef FORTRAN_FLOAT_FUNCTIONS_RETURN_DOUBLE
extern double slansf(
#else
extern float slansf(
#endif
    char   *norm,
    char   *transr,
    char   *uplo,
    ptrdiff_t *n,
    float  *a,
    float  *work
);

/* Source: slansp.f */
#define slansp FORTRAN_WRAPPER(slansp)
#ifdef FORTRAN_FLOAT_FUNCTIONS_RETURN_DOUBLE
extern double slansp(
#else
extern float slansp(
#endif
    char   *norm,
    char   *uplo,
    ptrdiff_t *n,
    float  *ap,
    float  *work
);

/* Source: slanst.f */
#define slanst FORTRAN_WRAPPER(slanst)
#ifdef FORTRAN_FLOAT_FUNCTIONS_RETURN_DOUBLE
extern double slanst(
#else
extern float slanst(
#endif
    char   *norm,
    ptrdiff_t *n,
    float  *d,
    float  *e
);

/* Source: slansy.f */
#define slansy FORTRAN_WRAPPER(slansy)
#ifdef FORTRAN_FLOAT_FUNCTIONS_RETURN_DOUBLE
extern double slansy(
#else
extern float slansy(
#endif
    char   *norm,
    char   *uplo,
    ptrdiff_t *n,
    float  *a,
    ptrdiff_t *lda,
    float  *work
);

/* Source: slantb.f */
#define slantb FORTRAN_WRAPPER(slantb)
#ifdef FORTRAN_FLOAT_FUNCTIONS_RETURN_DOUBLE
extern double slantb(
#else
extern float slantb(
#endif
    char   *norm,
    char   *uplo,
    char   *diag,
    ptrdiff_t *n,
    ptrdiff_t *k,
    float  *ab,
    ptrdiff_t *ldab,
    float  *work
);

/* Source: slantp.f */
#define slantp FORTRAN_WRAPPER(slantp)
#ifdef FORTRAN_FLOAT_FUNCTIONS_RETURN_DOUBLE
extern double slantp(
#else
extern float slantp(
#endif
    char   *norm,
    char   *uplo,
    char   *diag,
    ptrdiff_t *n,
    float  *ap,
    float  *work
);

/* Source: slantr.f */
#define slantr FORTRAN_WRAPPER(slantr)
#ifdef FORTRAN_FLOAT_FUNCTIONS_RETURN_DOUBLE
extern double slantr(
#else
extern float slantr(
#endif
    char   *norm,
    char   *uplo,
    char   *diag,
    ptrdiff_t *m,
    ptrdiff_t *n,
    float  *a,
    ptrdiff_t *lda,
    float  *work
);

/* Source: slanv2.f */
#define slanv2 FORTRAN_WRAPPER(slanv2)
extern void slanv2(
    float  *a,
    float  *b,
    float  *c,
    float  *d,
    float  *rt1r,
    float  *rt1i,
    float  *rt2r,
    float  *rt2i,
    float  *cs,
    float  *sn
);

/* Source: slapll.f */
#define slapll FORTRAN_WRAPPER(slapll)
extern void slapll(
    ptrdiff_t *n,
    float  *x,
    ptrdiff_t *incx,
    float  *y,
    ptrdiff_t *incy,
    float  *ssmin
);

/* Source: slapmt.f */
#define slapmt FORTRAN_WRAPPER(slapmt)
extern void slapmt(
    ptrdiff_t *forwrd,
    ptrdiff_t *m,
    ptrdiff_t *n,
    float  *x,
    ptrdiff_t *ldx,
    ptrdiff_t *k
);

/* Source: slapy2.f */
#define slapy2 FORTRAN_WRAPPER(slapy2)
#ifdef FORTRAN_FLOAT_FUNCTIONS_RETURN_DOUBLE
extern double slapy2(
#else
extern float slapy2(
#endif
    float  *x,
    float  *y
);

/* Source: slapy3.f */
#define slapy3 FORTRAN_WRAPPER(slapy3)
#ifdef FORTRAN_FLOAT_FUNCTIONS_RETURN_DOUBLE
extern double slapy3(
#else
extern float slapy3(
#endif
    float  *x,
    float  *y,
    float  *z
);

/* Source: slaqgb.f */
#define slaqgb FORTRAN_WRAPPER(slaqgb)
extern void slaqgb(
    ptrdiff_t *m,
    ptrdiff_t *n,
    ptrdiff_t *kl,
    ptrdiff_t *ku,
    float  *ab,
    ptrdiff_t *ldab,
    float  *r,
    float  *c,
    float  *rowcnd,
    float  *colcnd,
    float  *amax,
    char   *equed
);

/* Source: slaqge.f */
#define slaqge FORTRAN_WRAPPER(slaqge)
extern void slaqge(
    ptrdiff_t *m,
    ptrdiff_t *n,
    float  *a,
    ptrdiff_t *lda,
    float  *r,
    float  *c,
    float  *rowcnd,
    float  *colcnd,
    float  *amax,
    char   *equed
);

/* Source: slaqp2.f */
#define slaqp2 FORTRAN_WRAPPER(slaqp2)
extern void slaqp2(
    ptrdiff_t *m,
    ptrdiff_t *n,
    ptrdiff_t *offset,
    float  *a,
    ptrdiff_t *lda,
    ptrdiff_t *jpvt,
    float  *tau,
    float  *vn1,
    float  *vn2,
    float  *work
);

/* Source: slaqps.f */
#define slaqps FORTRAN_WRAPPER(slaqps)
extern void slaqps(
    ptrdiff_t *m,
    ptrdiff_t *n,
    ptrdiff_t *offset,
    ptrdiff_t *nb,
    ptrdiff_t *kb,
    float  *a,
    ptrdiff_t *lda,
    ptrdiff_t *jpvt,
    float  *tau,
    float  *vn1,
    float  *vn2,
    float  *auxv,
    float  *f,
    ptrdiff_t *ldf
);

/* Source: slaqr0.f */
#define slaqr0 FORTRAN_WRAPPER(slaqr0)
extern void slaqr0(
    ptrdiff_t *wantt,
    ptrdiff_t *wantz,
    ptrdiff_t *n,
    ptrdiff_t *ilo,
    ptrdiff_t *ihi,
    float  *h,
    ptrdiff_t *ldh,
    float  *wr,
    float  *wi,
    ptrdiff_t *iloz,
    ptrdiff_t *ihiz,
    float  *z,
    ptrdiff_t *ldz,
    float  *work,
    ptrdiff_t *lwork,
    ptrdiff_t *info
);

/* Source: slaqr1.f */
#define slaqr1 FORTRAN_WRAPPER(slaqr1)
extern void slaqr1(
    ptrdiff_t *n,
    float  *h,
    ptrdiff_t *ldh,
    float  *sr1,
    float  *si1,
    float  *sr2,
    float  *si2,
    float  *v
);

/* Source: slaqr2.f */
#define slaqr2 FORTRAN_WRAPPER(slaqr2)
extern void slaqr2(
    ptrdiff_t *wantt,
    ptrdiff_t *wantz,
    ptrdiff_t *n,
    ptrdiff_t *ktop,
    ptrdiff_t *kbot,
    ptrdiff_t *nw,
    float  *h,
    ptrdiff_t *ldh,
    ptrdiff_t *iloz,
    ptrdiff_t *ihiz,
    float  *z,
    ptrdiff_t *ldz,
    ptrdiff_t *ns,
    ptrdiff_t *nd,
    float  *sr,
    float  *si,
    float  *v,
    ptrdiff_t *ldv,
    ptrdiff_t *nh,
    float  *t,
    ptrdiff_t *ldt,
    ptrdiff_t *nv,
    float  *wv,
    ptrdiff_t *ldwv,
    float  *work,
    ptrdiff_t *lwork
);

/* Source: slaqr3.f */
#define slaqr3 FORTRAN_WRAPPER(slaqr3)
extern void slaqr3(
    ptrdiff_t *wantt,
    ptrdiff_t *wantz,
    ptrdiff_t *n,
    ptrdiff_t *ktop,
    ptrdiff_t *kbot,
    ptrdiff_t *nw,
    float  *h,
    ptrdiff_t *ldh,
    ptrdiff_t *iloz,
    ptrdiff_t *ihiz,
    float  *z,
    ptrdiff_t *ldz,
    ptrdiff_t *ns,
    ptrdiff_t *nd,
    float  *sr,
    float  *si,
    float  *v,
    ptrdiff_t *ldv,
    ptrdiff_t *nh,
    float  *t,
    ptrdiff_t *ldt,
    ptrdiff_t *nv,
    float  *wv,
    ptrdiff_t *ldwv,
    float  *work,
    ptrdiff_t *lwork
);

/* Source: slaqr4.f */
#define slaqr4 FORTRAN_WRAPPER(slaqr4)
extern void slaqr4(
    ptrdiff_t *wantt,
    ptrdiff_t *wantz,
    ptrdiff_t *n,
    ptrdiff_t *ilo,
    ptrdiff_t *ihi,
    float  *h,
    ptrdiff_t *ldh,
    float  *wr,
    float  *wi,
    ptrdiff_t *iloz,
    ptrdiff_t *ihiz,
    float  *z,
    ptrdiff_t *ldz,
    float  *work,
    ptrdiff_t *lwork,
    ptrdiff_t *info
);

/* Source: slaqr5.f */
#define slaqr5 FORTRAN_WRAPPER(slaqr5)
extern void slaqr5(
    ptrdiff_t *wantt,
    ptrdiff_t *wantz,
    ptrdiff_t *kacc22,
    ptrdiff_t *n,
    ptrdiff_t *ktop,
    ptrdiff_t *kbot,
    ptrdiff_t *nshfts,
    float  *sr,
    float  *si,
    float  *h,
    ptrdiff_t *ldh,
    ptrdiff_t *iloz,
    ptrdiff_t *ihiz,
    float  *z,
    ptrdiff_t *ldz,
    float  *v,
    ptrdiff_t *ldv,
    float  *u,
    ptrdiff_t *ldu,
    ptrdiff_t *nv,
    float  *wv,
    ptrdiff_t *ldwv,
    ptrdiff_t *nh,
    float  *wh,
    ptrdiff_t *ldwh
);

/* Source: slaqsb.f */
#define slaqsb FORTRAN_WRAPPER(slaqsb)
extern void slaqsb(
    char   *uplo,
    ptrdiff_t *n,
    ptrdiff_t *kd,
    float  *ab,
    ptrdiff_t *ldab,
    float  *s,
    float  *scond,
    float  *amax,
    char   *equed
);

/* Source: slaqsp.f */
#define slaqsp FORTRAN_WRAPPER(slaqsp)
extern void slaqsp(
    char   *uplo,
    ptrdiff_t *n,
    float  *ap,
    float  *s,
    float  *scond,
    float  *amax,
    char   *equed
);

/* Source: slaqsy.f */
#define slaqsy FORTRAN_WRAPPER(slaqsy)
extern void slaqsy(
    char   *uplo,
    ptrdiff_t *n,
    float  *a,
    ptrdiff_t *lda,
    float  *s,
    float  *scond,
    float  *amax,
    char   *equed
);

/* Source: slaqtr.f */
#define slaqtr FORTRAN_WRAPPER(slaqtr)
extern void slaqtr(
    ptrdiff_t *ltran,
    ptrdiff_t *lreal,
    ptrdiff_t *n,
    float  *t,
    ptrdiff_t *ldt,
    float  *b,
    float  *w,
    float  *scale,
    float  *x,
    float  *work,
    ptrdiff_t *info
);

/* Source: slar1v.f */
#define slar1v FORTRAN_WRAPPER(slar1v)
extern void slar1v(
    ptrdiff_t *n,
    ptrdiff_t *b1,
    ptrdiff_t *bn,
    float  *lambda,
    float  *d,
    float  *l,
    float  *ld,
    float  *lld,
    float  *pivmin,
    float  *gaptol,
    float  *z,
    ptrdiff_t *wantnc,
    ptrdiff_t *negcnt,
    float  *ztz,
    float  *mingma,
    ptrdiff_t *r,
    ptrdiff_t *isuppz,
    float  *nrminv,
    float  *resid,
    float  *rqcorr,
    float  *work
);

/* Source: slar2v.f */
#define slar2v FORTRAN_WRAPPER(slar2v)
extern void slar2v(
    ptrdiff_t *n,
    float  *x,
    float  *y,
    float  *z,
    ptrdiff_t *incx,
    float  *c,
    float  *s,
    ptrdiff_t *incc
);

/* Source: slarf.f */
#define slarf FORTRAN_WRAPPER(slarf)
extern void slarf(
    char   *side,
    ptrdiff_t *m,
    ptrdiff_t *n,
    float  *v,
    ptrdiff_t *incv,
    float  *tau,
    float  *c,
    ptrdiff_t *ldc,
    float  *work
);

/* Source: slarfb.f */
#define slarfb FORTRAN_WRAPPER(slarfb)
extern void slarfb(
    char   *side,
    char   *trans,
    char   *direct,
    char   *storev,
    ptrdiff_t *m,
    ptrdiff_t *n,
    ptrdiff_t *k,
    float  *v,
    ptrdiff_t *ldv,
    float  *t,
    ptrdiff_t *ldt,
    float  *c,
    ptrdiff_t *ldc,
    float  *work,
    ptrdiff_t *ldwork
);

/* Source: slarfg.f */
#define slarfg FORTRAN_WRAPPER(slarfg)
extern void slarfg(
    ptrdiff_t *n,
    float  *alpha,
    float  *x,
    ptrdiff_t *incx,
    float  *tau
);

/* Source: slarfgp.f */
#define slarfgp FORTRAN_WRAPPER(slarfgp)
extern void slarfgp(
    ptrdiff_t *n,
    float  *alpha,
    float  *x,
    ptrdiff_t *incx,
    float  *tau
);

/* Source: slarft.f */
#define slarft FORTRAN_WRAPPER(slarft)
extern void slarft(
    char   *direct,
    char   *storev,
    ptrdiff_t *n,
    ptrdiff_t *k,
    float  *v,
    ptrdiff_t *ldv,
    float  *tau,
    float  *t,
    ptrdiff_t *ldt
);

/* Source: slarfx.f */
#define slarfx FORTRAN_WRAPPER(slarfx)
extern void slarfx(
    char   *side,
    ptrdiff_t *m,
    ptrdiff_t *n,
    float  *v,
    float  *tau,
    float  *c,
    ptrdiff_t *ldc,
    float  *work
);

/* Source: slargv.f */
#define slargv FORTRAN_WRAPPER(slargv)
extern void slargv(
    ptrdiff_t *n,
    float  *x,
    ptrdiff_t *incx,
    float  *y,
    ptrdiff_t *incy,
    float  *c,
    ptrdiff_t *incc
);

/* Source: slarnv.f */
#define slarnv FORTRAN_WRAPPER(slarnv)
extern void slarnv(
    ptrdiff_t *idist,
    ptrdiff_t *iseed,
    ptrdiff_t *n,
    float  *x
);

/* Source: slarra.f */
#define slarra FORTRAN_WRAPPER(slarra)
extern void slarra(
    ptrdiff_t *n,
    float  *d,
    float  *e,
    float  *e2,
    float  *spltol,
    float  *tnrm,
    ptrdiff_t *nsplit,
    ptrdiff_t *isplit,
    ptrdiff_t *info
);

/* Source: slarrb.f */
#define slarrb FORTRAN_WRAPPER(slarrb)
extern void slarrb(
    ptrdiff_t *n,
    float  *d,
    float  *lld,
    ptrdiff_t *ifirst,
    ptrdiff_t *ilast,
    float  *rtol1,
    float  *rtol2,
    ptrdiff_t *offset,
    float  *w,
    float  *wgap,
    float  *werr,
    float  *work,
    ptrdiff_t *iwork,
    float  *pivmin,
    float  *spdiam,
    ptrdiff_t *twist,
    ptrdiff_t *info
);

/* Source: slarrc.f */
#define slarrc FORTRAN_WRAPPER(slarrc)
extern void slarrc(
    char   *jobt,
    ptrdiff_t *n,
    float  *vl,
    float  *vu,
    float  *d,
    float  *e,
    float  *pivmin,
    ptrdiff_t *eigcnt,
    ptrdiff_t *lcnt,
    ptrdiff_t *rcnt,
    ptrdiff_t *info
);

/* Source: slarrd.f */
#define slarrd FORTRAN_WRAPPER(slarrd)
extern void slarrd(
    char   *range,
    char   *order,
    ptrdiff_t *n,
    float  *vl,
    float  *vu,
    ptrdiff_t *il,
    ptrdiff_t *iu,
    float  *gers,
    float  *reltol,
    float  *d,
    float  *e,
    float  *e2,
    float  *pivmin,
    ptrdiff_t *nsplit,
    ptrdiff_t *isplit,
    ptrdiff_t *m,
    float  *w,
    float  *werr,
    float  *wl,
    float  *wu,
    ptrdiff_t *iblock,
    ptrdiff_t *indexw,
    float  *work,
    ptrdiff_t *iwork,
    ptrdiff_t *info
);

/* Source: slarre.f */
#define slarre FORTRAN_WRAPPER(slarre)
extern void slarre(
    char   *range,
    ptrdiff_t *n,
    float  *vl,
    float  *vu,
    ptrdiff_t *il,
    ptrdiff_t *iu,
    float  *d,
    float  *e,
    float  *e2,
    float  *rtol1,
    float  *rtol2,
    float  *spltol,
    ptrdiff_t *nsplit,
    ptrdiff_t *isplit,
    ptrdiff_t *m,
    float  *w,
    float  *werr,
    float  *wgap,
    ptrdiff_t *iblock,
    ptrdiff_t *indexw,
    float  *gers,
    float  *pivmin,
    float  *work,
    ptrdiff_t *iwork,
    ptrdiff_t *info
);

/* Source: slarrf.f */
#define slarrf FORTRAN_WRAPPER(slarrf)
extern void slarrf(
    ptrdiff_t *n,
    float  *d,
    float  *l,
    float  *ld,
    ptrdiff_t *clstrt,
    ptrdiff_t *clend,
    float  *w,
    float  *wgap,
    float  *werr,
    float  *spdiam,
    float  *clgapl,
    float  *clgapr,
    float  *pivmin,
    float  *sigma,
    float  *dplus,
    float  *lplus,
    float  *work,
    ptrdiff_t *info
);

/* Source: slarrj.f */
#define slarrj FORTRAN_WRAPPER(slarrj)
extern void slarrj(
    ptrdiff_t *n,
    float  *d,
    float  *e2,
    ptrdiff_t *ifirst,
    ptrdiff_t *ilast,
    float  *rtol,
    ptrdiff_t *offset,
    float  *w,
    float  *werr,
    float  *work,
    ptrdiff_t *iwork,
    float  *pivmin,
    float  *spdiam,
    ptrdiff_t *info
);

/* Source: slarrk.f */
#define slarrk FORTRAN_WRAPPER(slarrk)
extern void slarrk(
    ptrdiff_t *n,
    ptrdiff_t *iw,
    float  *gl,
    float  *gu,
    float  *d,
    float  *e2,
    float  *pivmin,
    float  *reltol,
    float  *w,
    float  *werr,
    ptrdiff_t *info
);

/* Source: slarrr.f */
#define slarrr FORTRAN_WRAPPER(slarrr)
extern void slarrr(
    ptrdiff_t *n,
    float  *d,
    float  *e,
    ptrdiff_t *info
);

/* Source: slarrv.f */
#define slarrv FORTRAN_WRAPPER(slarrv)
extern void slarrv(
    ptrdiff_t *n,
    float  *vl,
    float  *vu,
    float  *d,
    float  *l,
    float  *pivmin,
    ptrdiff_t *isplit,
    ptrdiff_t *m,
    ptrdiff_t *dol,
    ptrdiff_t *dou,
    float  *minrgp,
    float  *rtol1,
    float  *rtol2,
    float  *w,
    float  *werr,
    float  *wgap,
    ptrdiff_t *iblock,
    ptrdiff_t *indexw,
    float  *gers,
    float  *z,
    ptrdiff_t *ldz,
    ptrdiff_t *isuppz,
    float  *work,
    ptrdiff_t *iwork,
    ptrdiff_t *info
);

/* Source: slartg.f */
#define slartg FORTRAN_WRAPPER(slartg)
extern void slartg(
    float  *f,
    float  *g,
    float  *cs,
    float  *sn,
    float  *r
);

/* Source: slartv.f */
#define slartv FORTRAN_WRAPPER(slartv)
extern void slartv(
    ptrdiff_t *n,
    float  *x,
    ptrdiff_t *incx,
    float  *y,
    ptrdiff_t *incy,
    float  *c,
    float  *s,
    ptrdiff_t *incc
);

/* Source: slaruv.f */
#define slaruv FORTRAN_WRAPPER(slaruv)
extern void slaruv(
    ptrdiff_t *iseed,
    ptrdiff_t *n,
    float  *x
);

/* Source: slarz.f */
#define slarz FORTRAN_WRAPPER(slarz)
extern void slarz(
    char   *side,
    ptrdiff_t *m,
    ptrdiff_t *n,
    ptrdiff_t *l,
    float  *v,
    ptrdiff_t *incv,
    float  *tau,
    float  *c,
    ptrdiff_t *ldc,
    float  *work
);

/* Source: slarzb.f */
#define slarzb FORTRAN_WRAPPER(slarzb)
extern void slarzb(
    char   *side,
    char   *trans,
    char   *direct,
    char   *storev,
    ptrdiff_t *m,
    ptrdiff_t *n,
    ptrdiff_t *k,
    ptrdiff_t *l,
    float  *v,
    ptrdiff_t *ldv,
    float  *t,
    ptrdiff_t *ldt,
    float  *c,
    ptrdiff_t *ldc,
    float  *work,
    ptrdiff_t *ldwork
);

/* Source: slarzt.f */
#define slarzt FORTRAN_WRAPPER(slarzt)
extern void slarzt(
    char   *direct,
    char   *storev,
    ptrdiff_t *n,
    ptrdiff_t *k,
    float  *v,
    ptrdiff_t *ldv,
    float  *tau,
    float  *t,
    ptrdiff_t *ldt
);

/* Source: slas2.f */
#define slas2 FORTRAN_WRAPPER(slas2)
extern void slas2(
    float  *f,
    float  *g,
    float  *h,
    float  *ssmin,
    float  *ssmax
);

/* Source: slascl.f */
#define slascl FORTRAN_WRAPPER(slascl)
extern void slascl(
    char   *type,
    ptrdiff_t *kl,
    ptrdiff_t *ku,
    float  *cfrom,
    float  *cto,
    ptrdiff_t *m,
    ptrdiff_t *n,
    float  *a,
    ptrdiff_t *lda,
    ptrdiff_t *info
);

/* Source: slasd0.f */
#define slasd0 FORTRAN_WRAPPER(slasd0)
extern void slasd0(
    ptrdiff_t *n,
    ptrdiff_t *sqre,
    float  *d,
    float  *e,
    float  *u,
    ptrdiff_t *ldu,
    float  *vt,
    ptrdiff_t *ldvt,
    ptrdiff_t *smlsiz,
    ptrdiff_t *iwork,
    float  *work,
    ptrdiff_t *info
);

/* Source: slasd1.f */
#define slasd1 FORTRAN_WRAPPER(slasd1)
extern void slasd1(
    ptrdiff_t *nl,
    ptrdiff_t *nr,
    ptrdiff_t *sqre,
    float  *d,
    float  *alpha,
    float  *beta,
    float  *u,
    ptrdiff_t *ldu,
    float  *vt,
    ptrdiff_t *ldvt,
    ptrdiff_t *idxq,
    ptrdiff_t *iwork,
    float  *work,
    ptrdiff_t *info
);

/* Source: slasd2.f */
#define slasd2 FORTRAN_WRAPPER(slasd2)
extern void slasd2(
    ptrdiff_t *nl,
    ptrdiff_t *nr,
    ptrdiff_t *sqre,
    ptrdiff_t *k,
    float  *d,
    float  *z,
    float  *alpha,
    float  *beta,
    float  *u,
    ptrdiff_t *ldu,
    float  *vt,
    ptrdiff_t *ldvt,
    float  *dsigma,
    float  *u2,
    ptrdiff_t *ldu2,
    float  *vt2,
    ptrdiff_t *ldvt2,
    ptrdiff_t *idxp,
    ptrdiff_t *idx,
    ptrdiff_t *idxc,
    ptrdiff_t *idxq,
    ptrdiff_t *coltyp,
    ptrdiff_t *info
);

/* Source: slasd3.f */
#define slasd3 FORTRAN_WRAPPER(slasd3)
extern void slasd3(
    ptrdiff_t *nl,
    ptrdiff_t *nr,
    ptrdiff_t *sqre,
    ptrdiff_t *k,
    float  *d,
    float  *q,
    ptrdiff_t *ldq,
    float  *dsigma,
    float  *u,
    ptrdiff_t *ldu,
    float  *u2,
    ptrdiff_t *ldu2,
    float  *vt,
    ptrdiff_t *ldvt,
    float  *vt2,
    ptrdiff_t *ldvt2,
    ptrdiff_t *idxc,
    ptrdiff_t *ctot,
    float  *z,
    ptrdiff_t *info
);

/* Source: slasd4.f */
#define slasd4 FORTRAN_WRAPPER(slasd4)
extern void slasd4(
    ptrdiff_t *n,
    ptrdiff_t *i,
    float  *d,
    float  *z,
    float  *delta,
    float  *rho,
    float  *sigma,
    float  *work,
    ptrdiff_t *info
);

/* Source: slasd5.f */
#define slasd5 FORTRAN_WRAPPER(slasd5)
extern void slasd5(
    ptrdiff_t *i,
    float  *d,
    float  *z,
    float  *delta,
    float  *rho,
    float  *dsigma,
    float  *work
);

/* Source: slasd6.f */
#define slasd6 FORTRAN_WRAPPER(slasd6)
extern void slasd6(
    ptrdiff_t *icompq,
    ptrdiff_t *nl,
    ptrdiff_t *nr,
    ptrdiff_t *sqre,
    float  *d,
    float  *vf,
    float  *vl,
    float  *alpha,
    float  *beta,
    ptrdiff_t *idxq,
    ptrdiff_t *perm,
    ptrdiff_t *givptr,
    ptrdiff_t *givcol,
    ptrdiff_t *ldgcol,
    float  *givnum,
    ptrdiff_t *ldgnum,
    float  *poles,
    float  *difl,
    float  *difr,
    float  *z,
    ptrdiff_t *k,
    float  *c,
    float  *s,
    float  *work,
    ptrdiff_t *iwork,
    ptrdiff_t *info
);

/* Source: slasd7.f */
#define slasd7 FORTRAN_WRAPPER(slasd7)
extern void slasd7(
    ptrdiff_t *icompq,
    ptrdiff_t *nl,
    ptrdiff_t *nr,
    ptrdiff_t *sqre,
    ptrdiff_t *k,
    float  *d,
    float  *z,
    float  *zw,
    float  *vf,
    float  *vfw,
    float  *vl,
    float  *vlw,
    float  *alpha,
    float  *beta,
    float  *dsigma,
    ptrdiff_t *idx,
    ptrdiff_t *idxp,
    ptrdiff_t *idxq,
    ptrdiff_t *perm,
    ptrdiff_t *givptr,
    ptrdiff_t *givcol,
    ptrdiff_t *ldgcol,
    float  *givnum,
    ptrdiff_t *ldgnum,
    float  *c,
    float  *s,
    ptrdiff_t *info
);

/* Source: slasd8.f */
#define slasd8 FORTRAN_WRAPPER(slasd8)
extern void slasd8(
    ptrdiff_t *icompq,
    ptrdiff_t *k,
    float  *d,
    float  *z,
    float  *vf,
    float  *vl,
    float  *difl,
    float  *difr,
    ptrdiff_t *lddifr,
    float  *dsigma,
    float  *work,
    ptrdiff_t *info
);

/* Source: slasda.f */
#define slasda FORTRAN_WRAPPER(slasda)
extern void slasda(
    ptrdiff_t *icompq,
    ptrdiff_t *smlsiz,
    ptrdiff_t *n,
    ptrdiff_t *sqre,
    float  *d,
    float  *e,
    float  *u,
    ptrdiff_t *ldu,
    float  *vt,
    ptrdiff_t *k,
    float  *difl,
    float  *difr,
    float  *z,
    float  *poles,
    ptrdiff_t *givptr,
    ptrdiff_t *givcol,
    ptrdiff_t *ldgcol,
    ptrdiff_t *perm,
    float  *givnum,
    float  *c,
    float  *s,
    float  *work,
    ptrdiff_t *iwork,
    ptrdiff_t *info
);

/* Source: slasdq.f */
#define slasdq FORTRAN_WRAPPER(slasdq)
extern void slasdq(
    char   *uplo,
    ptrdiff_t *sqre,
    ptrdiff_t *n,
    ptrdiff_t *ncvt,
    ptrdiff_t *nru,
    ptrdiff_t *ncc,
    float  *d,
    float  *e,
    float  *vt,
    ptrdiff_t *ldvt,
    float  *u,
    ptrdiff_t *ldu,
    float  *c,
    ptrdiff_t *ldc,
    float  *work,
    ptrdiff_t *info
);

/* Source: slasdt.f */
#define slasdt FORTRAN_WRAPPER(slasdt)
extern void slasdt(
    ptrdiff_t *n,
    ptrdiff_t *lvl,
    ptrdiff_t *nd,
    ptrdiff_t *inode,
    ptrdiff_t *ndiml,
    ptrdiff_t *ndimr,
    ptrdiff_t *msub
);

/* Source: slaset.f */
#define slaset FORTRAN_WRAPPER(slaset)
extern void slaset(
    char   *uplo,
    ptrdiff_t *m,
    ptrdiff_t *n,
    float  *alpha,
    float  *beta,
    float  *a,
    ptrdiff_t *lda
);

/* Source: slasq1.f */
#define slasq1 FORTRAN_WRAPPER(slasq1)
extern void slasq1(
    ptrdiff_t *n,
    float  *d,
    float  *e,
    float  *work,
    ptrdiff_t *info
);

/* Source: slasq2.f */
#define slasq2 FORTRAN_WRAPPER(slasq2)
extern void slasq2(
    ptrdiff_t *n,
    float  *z,
    ptrdiff_t *info
);

/* Source: slasq3.f */
#define slasq3 FORTRAN_WRAPPER(slasq3)
extern void slasq3(
    ptrdiff_t *i0,
    ptrdiff_t *n0,
    float  *z,
    ptrdiff_t *pp,
    float  *dmin,
    float  *sigma,
    float  *desig,
    float  *qmax,
    ptrdiff_t *nfail,
    ptrdiff_t *iter,
    ptrdiff_t *ndiv,
    ptrdiff_t *ieee,
    ptrdiff_t *ttype,
    float  *dmin1,
    float  *dmin2,
    float  *dn,
    float  *dn1,
    float  *dn2,
    float  *g,
    float  *tau
);

/* Source: slasq4.f */
#define slasq4 FORTRAN_WRAPPER(slasq4)
extern void slasq4(
    ptrdiff_t *i0,
    ptrdiff_t *n0,
    float  *z,
    ptrdiff_t *pp,
    ptrdiff_t *n0in,
    float  *dmin,
    float  *dmin1,
    float  *dmin2,
    float  *dn,
    float  *dn1,
    float  *dn2,
    float  *tau,
    ptrdiff_t *ttype,
    float  *g
);

/* Source: slasq5.f */
#define slasq5 FORTRAN_WRAPPER(slasq5)
extern void slasq5(
    ptrdiff_t *i0,
    ptrdiff_t *n0,
    float  *z,
    ptrdiff_t *pp,
    float  *tau,
    float  *dmin,
    float  *dmin1,
    float  *dmin2,
    float  *dn,
    float  *dnm1,
    float  *dnm2,
    ptrdiff_t *ieee
);

/* Source: slasq6.f */
#define slasq6 FORTRAN_WRAPPER(slasq6)
extern void slasq6(
    ptrdiff_t *i0,
    ptrdiff_t *n0,
    float  *z,
    ptrdiff_t *pp,
    float  *dmin,
    float  *dmin1,
    float  *dmin2,
    float  *dn,
    float  *dnm1,
    float  *dnm2
);

/* Source: slasr.f */
#define slasr FORTRAN_WRAPPER(slasr)
extern void slasr(
    char   *side,
    char   *pivot,
    char   *direct,
    ptrdiff_t *m,
    ptrdiff_t *n,
    float  *c,
    float  *s,
    float  *a,
    ptrdiff_t *lda
);

/* Source: slasrt.f */
#define slasrt FORTRAN_WRAPPER(slasrt)
extern void slasrt(
    char   *id,
    ptrdiff_t *n,
    float  *d,
    ptrdiff_t *info
);

/* Source: slassq.f */
#define slassq FORTRAN_WRAPPER(slassq)
extern void slassq(
    ptrdiff_t *n,
    float  *x,
    ptrdiff_t *incx,
    float  *scale,
    float  *sumsq
);

/* Source: slasv2.f */
#define slasv2 FORTRAN_WRAPPER(slasv2)
extern void slasv2(
    float  *f,
    float  *g,
    float  *h,
    float  *ssmin,
    float  *ssmax,
    float  *snr,
    float  *csr,
    float  *snl,
    float  *csl
);

/* Source: slaswp.f */
#define slaswp FORTRAN_WRAPPER(slaswp)
extern void slaswp(
    ptrdiff_t *n,
    float  *a,
    ptrdiff_t *lda,
    ptrdiff_t *k1,
    ptrdiff_t *k2,
    ptrdiff_t *ipiv,
    ptrdiff_t *incx
);

/* Source: slasy2.f */
#define slasy2 FORTRAN_WRAPPER(slasy2)
extern void slasy2(
    ptrdiff_t *ltranl,
    ptrdiff_t *ltranr,
    ptrdiff_t *isgn,
    ptrdiff_t *n1,
    ptrdiff_t *n2,
    float  *tl,
    ptrdiff_t *ldtl,
    float  *tr,
    ptrdiff_t *ldtr,
    float  *b,
    ptrdiff_t *ldb,
    float  *scale,
    float  *x,
    ptrdiff_t *ldx,
    float  *xnorm,
    ptrdiff_t *info
);

/* Source: slasyf.f */
#define slasyf FORTRAN_WRAPPER(slasyf)
extern void slasyf(
    char   *uplo,
    ptrdiff_t *n,
    ptrdiff_t *nb,
    ptrdiff_t *kb,
    float  *a,
    ptrdiff_t *lda,
    ptrdiff_t *ipiv,
    float  *w,
    ptrdiff_t *ldw,
    ptrdiff_t *info
);

/* Source: slatbs.f */
#define slatbs FORTRAN_WRAPPER(slatbs)
extern void slatbs(
    char   *uplo,
    char   *trans,
    char   *diag,
    char   *normin,
    ptrdiff_t *n,
    ptrdiff_t *kd,
    float  *ab,
    ptrdiff_t *ldab,
    float  *x,
    float  *scale,
    float  *cnorm,
    ptrdiff_t *info
);

/* Source: slatdf.f */
#define slatdf FORTRAN_WRAPPER(slatdf)
extern void slatdf(
    ptrdiff_t *ijob,
    ptrdiff_t *n,
    float  *z,
    ptrdiff_t *ldz,
    float  *rhs,
    float  *rdsum,
    float  *rdscal,
    ptrdiff_t *ipiv,
    ptrdiff_t *jpiv
);

/* Source: slatps.f */
#define slatps FORTRAN_WRAPPER(slatps)
extern void slatps(
    char   *uplo,
    char   *trans,
    char   *diag,
    char   *normin,
    ptrdiff_t *n,
    float  *ap,
    float  *x,
    float  *scale,
    float  *cnorm,
    ptrdiff_t *info
);

/* Source: slatrd.f */
#define slatrd FORTRAN_WRAPPER(slatrd)
extern void slatrd(
    char   *uplo,
    ptrdiff_t *n,
    ptrdiff_t *nb,
    float  *a,
    ptrdiff_t *lda,
    float  *e,
    float  *tau,
    float  *w,
    ptrdiff_t *ldw
);

/* Source: slatrs.f */
#define slatrs FORTRAN_WRAPPER(slatrs)
extern void slatrs(
    char   *uplo,
    char   *trans,
    char   *diag,
    char   *normin,
    ptrdiff_t *n,
    float  *a,
    ptrdiff_t *lda,
    float  *x,
    float  *scale,
    float  *cnorm,
    ptrdiff_t *info
);

/* Source: slatrz.f */
#define slatrz FORTRAN_WRAPPER(slatrz)
extern void slatrz(
    ptrdiff_t *m,
    ptrdiff_t *n,
    ptrdiff_t *l,
    float  *a,
    ptrdiff_t *lda,
    float  *tau,
    float  *work
);
```
